(* Logix 5000 project; controller Universal_Device_Info_AOI_V0_1 vendor 1 type 14 code 176 rev 32.11; software revision 32.00; part 3 of 10 *)

           TBEN_L4_8IOL:I.Data[62].11   // IO-Link Port 4 - Input data word 11 (INT bit11)
           TBEN_L4_8IOL:I.Data[62].12   // IO-Link Port 4 - Input data word 11 (INT bit12)
           TBEN_L4_8IOL:I.Data[62].13   // IO-Link Port 4 - Input data word 11 (INT bit13)
           TBEN_L4_8IOL:I.Data[62].14   // IO-Link Port 4 - Input data word 11 (INT bit14)
           TBEN_L4_8IOL:I.Data[62].15   // IO-Link Port 4 - Input data word 11 (INT bit15)
           TBEN_L4_8IOL:I.Data[62].2   // IO-Link Port 4 - Input data word 11 (INT bit2)
           TBEN_L4_8IOL:I.Data[62].3   // IO-Link Port 4 - Input data word 11 (INT bit3)
           TBEN_L4_8IOL:I.Data[62].4   // IO-Link Port 4 - Input data word 11 (INT bit4)
           TBEN_L4_8IOL:I.Data[62].5   // IO-Link Port 4 - Input data word 11 (INT bit5)
           TBEN_L4_8IOL:I.Data[62].6   // IO-Link Port 4 - Input data word 11 (INT bit6)
           TBEN_L4_8IOL:I.Data[62].7   // IO-Link Port 4 - Input data word 11 (INT bit7)
           TBEN_L4_8IOL:I.Data[62].8   // IO-Link Port 4 - Input data word 11 (INT bit8)
           TBEN_L4_8IOL:I.Data[62].9   // IO-Link Port 4 - Input data word 11 (INT bit9)
           TBEN_L4_8IOL:I.Data[63]   // IO-Link Port 4 - Input data word 12
           TBEN_L4_8IOL:I.Data[63].0   // IO-Link Port 4 - Input data word 12 (INT bit0)
           TBEN_L4_8IOL:I.Data[63].1   // IO-Link Port 4 - Input data word 12 (INT bit1)
           TBEN_L4_8IOL:I.Data[63].10   // IO-Link Port 4 - Input data word 12 (INT bit10)
           TBEN_L4_8IOL:I.Data[63].11   // IO-Link Port 4 - Input data word 12 (INT bit11)
           TBEN_L4_8IOL:I.Data[63].12   // IO-Link Port 4 - Input data word 12 (INT bit12)
           TBEN_L4_8IOL:I.Data[63].13   // IO-Link Port 4 - Input data word 12 (INT bit13)
           TBEN_L4_8IOL:I.Data[63].14   // IO-Link Port 4 - Input data word 12 (INT bit14)
           TBEN_L4_8IOL:I.Data[63].15   // IO-Link Port 4 - Input data word 12 (INT bit15)
           TBEN_L4_8IOL:I.Data[63].2   // IO-Link Port 4 - Input data word 12 (INT bit2)
           TBEN_L4_8IOL:I.Data[63].3   // IO-Link Port 4 - Input data word 12 (INT bit3)
           TBEN_L4_8IOL:I.Data[63].4   // IO-Link Port 4 - Input data word 12 (INT bit4)
           TBEN_L4_8IOL:I.Data[63].5   // IO-Link Port 4 - Input data word 12 (INT bit5)
           TBEN_L4_8IOL:I.Data[63].6   // IO-Link Port 4 - Input data word 12 (INT bit6)
           TBEN_L4_8IOL:I.Data[63].7   // IO-Link Port 4 - Input data word 12 (INT bit7)
           TBEN_L4_8IOL:I.Data[63].8   // IO-Link Port 4 - Input data word 12 (INT bit8)
           TBEN_L4_8IOL:I.Data[63].9   // IO-Link Port 4 - Input data word 12 (INT bit9)
           TBEN_L4_8IOL:I.Data[64]   // IO-Link Port 4 - Input data word 13
           TBEN_L4_8IOL:I.Data[64].0   // IO-Link Port 4 - Input data word 13 (INT bit0)
           TBEN_L4_8IOL:I.Data[64].1   // IO-Link Port 4 - Input data word 13 (INT bit1)
           TBEN_L4_8IOL:I.Data[64].10   // IO-Link Port 4 - Input data word 13 (INT bit10)
           TBEN_L4_8IOL:I.Data[64].11   // IO-Link Port 4 - Input data word 13 (INT bit11)
           TBEN_L4_8IOL:I.Data[64].12   // IO-Link Port 4 - Input data word 13 (INT bit12)
           TBEN_L4_8IOL:I.Data[64].13   // IO-Link Port 4 - Input data word 13 (INT bit13)
           TBEN_L4_8IOL:I.Data[64].14   // IO-Link Port 4 - Input data word 13 (INT bit14)
           TBEN_L4_8IOL:I.Data[64].15   // IO-Link Port 4 - Input data word 13 (INT bit15)
           TBEN_L4_8IOL:I.Data[64].2   // IO-Link Port 4 - Input data word 13 (INT bit2)
           TBEN_L4_8IOL:I.Data[64].3   // IO-Link Port 4 - Input data word 13 (INT bit3)
           TBEN_L4_8IOL:I.Data[64].4   // IO-Link Port 4 - Input data word 13 (INT bit4)
           TBEN_L4_8IOL:I.Data[64].5   // IO-Link Port 4 - Input data word 13 (INT bit5)
           TBEN_L4_8IOL:I.Data[64].6   // IO-Link Port 4 - Input data word 13 (INT bit6)
           TBEN_L4_8IOL:I.Data[64].7   // IO-Link Port 4 - Input data word 13 (INT bit7)
           TBEN_L4_8IOL:I.Data[64].8   // IO-Link Port 4 - Input data word 13 (INT bit8)
           TBEN_L4_8IOL:I.Data[64].9   // IO-Link Port 4 - Input data word 13 (INT bit9)
           TBEN_L4_8IOL:I.Data[65]   // IO-Link Port 4 - Input data word 14
           TBEN_L4_8IOL:I.Data[65].0   // IO-Link Port 4 - Input data word 14 (INT bit0)
           TBEN_L4_8IOL:I.Data[65].1   // IO-Link Port 4 - Input data word 14 (INT bit1)
           TBEN_L4_8IOL:I.Data[65].10   // IO-Link Port 4 - Input data word 14 (INT bit10)
           TBEN_L4_8IOL:I.Data[65].11   // IO-Link Port 4 - Input data word 14 (INT bit11)
           TBEN_L4_8IOL:I.Data[65].12   // IO-Link Port 4 - Input data word 14 (INT bit12)
           TBEN_L4_8IOL:I.Data[65].13   // IO-Link Port 4 - Input data word 14 (INT bit13)
           TBEN_L4_8IOL:I.Data[65].14   // IO-Link Port 4 - Input data word 14 (INT bit14)
           TBEN_L4_8IOL:I.Data[65].15   // IO-Link Port 4 - Input data word 14 (INT bit15)
           TBEN_L4_8IOL:I.Data[65].2   // IO-Link Port 4 - Input data word 14 (INT bit2)
           TBEN_L4_8IOL:I.Data[65].3   // IO-Link Port 4 - Input data word 14 (INT bit3)
           TBEN_L4_8IOL:I.Data[65].4   // IO-Link Port 4 - Input data word 14 (INT bit4)
           TBEN_L4_8IOL:I.Data[65].5   // IO-Link Port 4 - Input data word 14 (INT bit5)
           TBEN_L4_8IOL:I.Data[65].6   // IO-Link Port 4 - Input data word 14 (INT bit6)
           TBEN_L4_8IOL:I.Data[65].7   // IO-Link Port 4 - Input data word 14 (INT bit7)
           TBEN_L4_8IOL:I.Data[65].8   // IO-Link Port 4 - Input data word 14 (INT bit8)
           TBEN_L4_8IOL:I.Data[65].9   // IO-Link Port 4 - Input data word 14 (INT bit9)
           TBEN_L4_8IOL:I.Data[66]   // IO-Link Port 4 - Input data word 15
           TBEN_L4_8IOL:I.Data[66].0   // IO-Link Port 4 - Input data word 15 (INT bit0)
           TBEN_L4_8IOL:I.Data[66].1   // IO-Link Port 4 - Input data word 15 (INT bit1)
           TBEN_L4_8IOL:I.Data[66].10   // IO-Link Port 4 - Input data word 15 (INT bit10)
           TBEN_L4_8IOL:I.Data[66].11   // IO-Link Port 4 - Input data word 15 (INT bit11)
           TBEN_L4_8IOL:I.Data[66].12   // IO-Link Port 4 - Input data word 15 (INT bit12)
           TBEN_L4_8IOL:I.Data[66].13   // IO-Link Port 4 - Input data word 15 (INT bit13)
           TBEN_L4_8IOL:I.Data[66].14   // IO-Link Port 4 - Input data word 15 (INT bit14)
           TBEN_L4_8IOL:I.Data[66].15   // IO-Link Port 4 - Input data word 15 (INT bit15)
           TBEN_L4_8IOL:I.Data[66].2   // IO-Link Port 4 - Input data word 15 (INT bit2)
           TBEN_L4_8IOL:I.Data[66].3   // IO-Link Port 4 - Input data word 15 (INT bit3)
           TBEN_L4_8IOL:I.Data[66].4   // IO-Link Port 4 - Input data word 15 (INT bit4)
           TBEN_L4_8IOL:I.Data[66].5   // IO-Link Port 4 - Input data word 15 (INT bit5)
           TBEN_L4_8IOL:I.Data[66].6   // IO-Link Port 4 - Input data word 15 (INT bit6)
           TBEN_L4_8IOL:I.Data[66].7   // IO-Link Port 4 - Input data word 15 (INT bit7)
           TBEN_L4_8IOL:I.Data[66].8   // IO-Link Port 4 - Input data word 15 (INT bit8)
           TBEN_L4_8IOL:I.Data[66].9   // IO-Link Port 4 - Input data word 15 (INT bit9)
           TBEN_L4_8IOL:I.Data[67]   // IO-Link Port 5 - Input data word 0
           TBEN_L4_8IOL:I.Data[67].0   // IO-Link Port 5 - Input data word 0 (INT bit0)
           TBEN_L4_8IOL:I.Data[67].1   // IO-Link Port 5 - Input data word 0 (INT bit1)
           TBEN_L4_8IOL:I.Data[67].10   // IO-Link Port 5 - Input data word 0 (INT bit10)
           TBEN_L4_8IOL:I.Data[67].11   // IO-Link Port 5 - Input data word 0 (INT bit11)
           TBEN_L4_8IOL:I.Data[67].12   // IO-Link Port 5 - Input data word 0 (INT bit12)
           TBEN_L4_8IOL:I.Data[67].13   // IO-Link Port 5 - Input data word 0 (INT bit13)
           TBEN_L4_8IOL:I.Data[67].14   // IO-Link Port 5 - Input data word 0 (INT bit14)
           TBEN_L4_8IOL:I.Data[67].15   // IO-Link Port 5 - Input data word 0 (INT bit15)
           TBEN_L4_8IOL:I.Data[67].2   // IO-Link Port 5 - Input data word 0 (INT bit2)
           TBEN_L4_8IOL:I.Data[67].3   // IO-Link Port 5 - Input data word 0 (INT bit3)
           TBEN_L4_8IOL:I.Data[67].4   // IO-Link Port 5 - Input data word 0 (INT bit4)
           TBEN_L4_8IOL:I.Data[67].5   // IO-Link Port 5 - Input data word 0 (INT bit5)
           TBEN_L4_8IOL:I.Data[67].6   // IO-Link Port 5 - Input data word 0 (INT bit6)
           TBEN_L4_8IOL:I.Data[67].7   // IO-Link Port 5 - Input data word 0 (INT bit7)
           TBEN_L4_8IOL:I.Data[67].8   // IO-Link Port 5 - Input data word 0 (INT bit8)
           TBEN_L4_8IOL:I.Data[67].9   // IO-Link Port 5 - Input data word 0 (INT bit9)
           TBEN_L4_8IOL:I.Data[68]   // IO-Link Port 5 - Input data word 1
           TBEN_L4_8IOL:I.Data[68].0   // IO-Link Port 5 - Input data word 1 (INT bit0)
           TBEN_L4_8IOL:I.Data[68].1   // IO-Link Port 5 - Input data word 1 (INT bit1)
           TBEN_L4_8IOL:I.Data[68].10   // IO-Link Port 5 - Input data word 1 (INT bit10)
           TBEN_L4_8IOL:I.Data[68].11   // IO-Link Port 5 - Input data word 1 (INT bit11)
           TBEN_L4_8IOL:I.Data[68].12   // IO-Link Port 5 - Input data word 1 (INT bit12)
           TBEN_L4_8IOL:I.Data[68].13   // IO-Link Port 5 - Input data word 1 (INT bit13)
           TBEN_L4_8IOL:I.Data[68].14   // IO-Link Port 5 - Input data word 1 (INT bit14)
           TBEN_L4_8IOL:I.Data[68].15   // IO-Link Port 5 - Input data word 1 (INT bit15)
           TBEN_L4_8IOL:I.Data[68].2   // IO-Link Port 5 - Input data word 1 (INT bit2)
           TBEN_L4_8IOL:I.Data[68].3   // IO-Link Port 5 - Input data word 1 (INT bit3)
           TBEN_L4_8IOL:I.Data[68].4   // IO-Link Port 5 - Input data word 1 (INT bit4)
           TBEN_L4_8IOL:I.Data[68].5   // IO-Link Port 5 - Input data word 1 (INT bit5)
           TBEN_L4_8IOL:I.Data[68].6   // IO-Link Port 5 - Input data word 1 (INT bit6)
           TBEN_L4_8IOL:I.Data[68].7   // IO-Link Port 5 - Input data word 1 (INT bit7)
           TBEN_L4_8IOL:I.Data[68].8   // IO-Link Port 5 - Input data word 1 (INT bit8)
           TBEN_L4_8IOL:I.Data[68].9   // IO-Link Port 5 - Input data word 1 (INT bit9)
           TBEN_L4_8IOL:I.Data[69]   // IO-Link Port 5 - Input data word 2
           TBEN_L4_8IOL:I.Data[69].0   // IO-Link Port 5 - Input data word 2 (INT bit0)
           TBEN_L4_8IOL:I.Data[69].1   // IO-Link Port 5 - Input data word 2 (INT bit1)
           TBEN_L4_8IOL:I.Data[69].10   // IO-Link Port 5 - Input data word 2 (INT bit10)
           TBEN_L4_8IOL:I.Data[69].11   // IO-Link Port 5 - Input data word 2 (INT bit11)
           TBEN_L4_8IOL:I.Data[69].12   // IO-Link Port 5 - Input data word 2 (INT bit12)
           TBEN_L4_8IOL:I.Data[69].13   // IO-Link Port 5 - Input data word 2 (INT bit13)
           TBEN_L4_8IOL:I.Data[69].14   // IO-Link Port 5 - Input data word 2 (INT bit14)
           TBEN_L4_8IOL:I.Data[69].15   // IO-Link Port 5 - Input data word 2 (INT bit15)
           TBEN_L4_8IOL:I.Data[69].2   // IO-Link Port 5 - Input data word 2 (INT bit2)
           TBEN_L4_8IOL:I.Data[69].3   // IO-Link Port 5 - Input data word 2 (INT bit3)
           TBEN_L4_8IOL:I.Data[69].4   // IO-Link Port 5 - Input data word 2 (INT bit4)
           TBEN_L4_8IOL:I.Data[69].5   // IO-Link Port 5 - Input data word 2 (INT bit5)
           TBEN_L4_8IOL:I.Data[69].6   // IO-Link Port 5 - Input data word 2 (INT bit6)
           TBEN_L4_8IOL:I.Data[69].7   // IO-Link Port 5 - Input data word 2 (INT bit7)
           TBEN_L4_8IOL:I.Data[69].8   // IO-Link Port 5 - Input data word 2 (INT bit8)
           TBEN_L4_8IOL:I.Data[69].9   // IO-Link Port 5 - Input data word 2 (INT bit9)
           TBEN_L4_8IOL:I.Data[6]   // IO-Link Port 1 - Input data word 3
           TBEN_L4_8IOL:I.Data[6].0   // IO-Link Port 1 - Input data word 3 (INT bit0)
           TBEN_L4_8IOL:I.Data[6].1   // IO-Link Port 1 - Input data word 3 (INT bit1)
           TBEN_L4_8IOL:I.Data[6].10   // IO-Link Port 1 - Input data word 3 (INT bit10)
           TBEN_L4_8IOL:I.Data[6].11   // IO-Link Port 1 - Input data word 3 (INT bit11)
           TBEN_L4_8IOL:I.Data[6].12   // IO-Link Port 1 - Input data word 3 (INT bit12)
           TBEN_L4_8IOL:I.Data[6].13   // IO-Link Port 1 - Input data word 3 (INT bit13)
           TBEN_L4_8IOL:I.Data[6].14   // IO-Link Port 1 - Input data word 3 (INT bit14)
           TBEN_L4_8IOL:I.Data[6].15   // IO-Link Port 1 - Input data word 3 (INT bit15)
           TBEN_L4_8IOL:I.Data[6].2   // IO-Link Port 1 - Input data word 3 (INT bit2)
           TBEN_L4_8IOL:I.Data[6].3   // IO-Link Port 1 - Input data word 3 (INT bit3)
           TBEN_L4_8IOL:I.Data[6].4   // IO-Link Port 1 - Input data word 3 (INT bit4)
           TBEN_L4_8IOL:I.Data[6].5   // IO-Link Port 1 - Input data word 3 (INT bit5)
           TBEN_L4_8IOL:I.Data[6].6   // IO-Link Port 1 - Input data word 3 (INT bit6)
           TBEN_L4_8IOL:I.Data[6].7   // IO-Link Port 1 - Input data word 3 (INT bit7)
           TBEN_L4_8IOL:I.Data[6].8   // IO-Link Port 1 - Input data word 3 (INT bit8)
           TBEN_L4_8IOL:I.Data[6].9   // IO-Link Port 1 - Input data word 3 (INT bit9)
           TBEN_L4_8IOL:I.Data[70]   // IO-Link Port 5 - Input data word 3
           TBEN_L4_8IOL:I.Data[70].0   // IO-Link Port 5 - Input data word 3 (INT bit0)
           TBEN_L4_8IOL:I.Data[70].1   // IO-Link Port 5 - Input data word 3 (INT bit1)
           TBEN_L4_8IOL:I.Data[70].10   // IO-Link Port 5 - Input data word 3 (INT bit10)
           TBEN_L4_8IOL:I.Data[70].11   // IO-Link Port 5 - Input data word 3 (INT bit11)
           TBEN_L4_8IOL:I.Data[70].12   // IO-Link Port 5 - Input data word 3 (INT bit12)
           TBEN_L4_8IOL:I.Data[70].13   // IO-Link Port 5 - Input data word 3 (INT bit13)
           TBEN_L4_8IOL:I.Data[70].14   // IO-Link Port 5 - Input data word 3 (INT bit14)
           TBEN_L4_8IOL:I.Data[70].15   // IO-Link Port 5 - Input data word 3 (INT bit15)
           TBEN_L4_8IOL:I.Data[70].2   // IO-Link Port 5 - Input data word 3 (INT bit2)
           TBEN_L4_8IOL:I.Data[70].3   // IO-Link Port 5 - Input data word 3 (INT bit3)
           TBEN_L4_8IOL:I.Data[70].4   // IO-Link Port 5 - Input data word 3 (INT bit4)
           TBEN_L4_8IOL:I.Data[70].5   // IO-Link Port 5 - Input data word 3 (INT bit5)
           TBEN_L4_8IOL:I.Data[70].6   // IO-Link Port 5 - Input data word 3 (INT bit6)
           TBEN_L4_8IOL:I.Data[70].7   // IO-Link Port 5 - Input data word 3 (INT bit7)
           TBEN_L4_8IOL:I.Data[70].8   // IO-Link Port 5 - Input data word 3 (INT bit8)
           TBEN_L4_8IOL:I.Data[70].9   // IO-Link Port 5 - Input data word 3 (INT bit9)
           TBEN_L4_8IOL:I.Data[71]   // IO-Link Port 5 - Input data word 4
           TBEN_L4_8IOL:I.Data[71].0   // IO-Link Port 5 - Input data word 4 (INT bit0)
           TBEN_L4_8IOL:I.Data[71].1   // IO-Link Port 5 - Input data word 4 (INT bit1)
           TBEN_L4_8IOL:I.Data[71].10   // IO-Link Port 5 - Input data word 4 (INT bit10)
           TBEN_L4_8IOL:I.Data[71].11   // IO-Link Port 5 - Input data word 4 (INT bit11)
           TBEN_L4_8IOL:I.Data[71].12   // IO-Link Port 5 - Input data word 4 (INT bit12)
           TBEN_L4_8IOL:I.Data[71].13   // IO-Link Port 5 - Input data word 4 (INT bit13)
           TBEN_L4_8IOL:I.Data[71].14   // IO-Link Port 5 - Input data word 4 (INT bit14)
           TBEN_L4_8IOL:I.Data[71].15   // IO-Link Port 5 - Input data word 4 (INT bit15)
           TBEN_L4_8IOL:I.Data[71].2   // IO-Link Port 5 - Input data word 4 (INT bit2)
           TBEN_L4_8IOL:I.Data[71].3   // IO-Link Port 5 - Input data word 4 (INT bit3)
           TBEN_L4_8IOL:I.Data[71].4   // IO-Link Port 5 - Input data word 4 (INT bit4)
           TBEN_L4_8IOL:I.Data[71].5   // IO-Link Port 5 - Input data word 4 (INT bit5)
           TBEN_L4_8IOL:I.Data[71].6   // IO-Link Port 5 - Input data word 4 (INT bit6)
           TBEN_L4_8IOL:I.Data[71].7   // IO-Link Port 5 - Input data word 4 (INT bit7)
           TBEN_L4_8IOL:I.Data[71].8   // IO-Link Port 5 - Input data word 4 (INT bit8)
           TBEN_L4_8IOL:I.Data[71].9   // IO-Link Port 5 - Input data word 4 (INT bit9)
           TBEN_L4_8IOL:I.Data[72]   // IO-Link Port 5 - Input data word 5
           TBEN_L4_8IOL:I.Data[72].0   // IO-Link Port 5 - Input data word 5 (INT bit0)
           TBEN_L4_8IOL:I.Data[72].1   // IO-Link Port 5 - Input data word 5 (INT bit1)
           TBEN_L4_8IOL:I.Data[72].10   // IO-Link Port 5 - Input data word 5 (INT bit10)
           TBEN_L4_8IOL:I.Data[72].11   // IO-Link Port 5 - Input data word 5 (INT bit11)
           TBEN_L4_8IOL:I.Data[72].12   // IO-Link Port 5 - Input data word 5 (INT bit12)
           TBEN_L4_8IOL:I.Data[72].13   // IO-Link Port 5 - Input data word 5 (INT bit13)
           TBEN_L4_8IOL:I.Data[72].14   // IO-Link Port 5 - Input data word 5 (INT bit14)
           TBEN_L4_8IOL:I.Data[72].15   // IO-Link Port 5 - Input data word 5 (INT bit15)
           TBEN_L4_8IOL:I.Data[72].2   // IO-Link Port 5 - Input data word 5 (INT bit2)
           TBEN_L4_8IOL:I.Data[72].3   // IO-Link Port 5 - Input data word 5 (INT bit3)
           TBEN_L4_8IOL:I.Data[72].4   // IO-Link Port 5 - Input data word 5 (INT bit4)
           TBEN_L4_8IOL:I.Data[72].5   // IO-Link Port 5 - Input data word 5 (INT bit5)
           TBEN_L4_8IOL:I.Data[72].6   // IO-Link Port 5 - Input data word 5 (INT bit6)
           TBEN_L4_8IOL:I.Data[72].7   // IO-Link Port 5 - Input data word 5 (INT bit7)
           TBEN_L4_8IOL:I.Data[72].8   // IO-Link Port 5 - Input data word 5 (INT bit8)
           TBEN_L4_8IOL:I.Data[72].9   // IO-Link Port 5 - Input data word 5 (INT bit9)
           TBEN_L4_8IOL:I.Data[73]   // IO-Link Port 5 - Input data word 6
           TBEN_L4_8IOL:I.Data[73].0   // IO-Link Port 5 - Input data word 6 (INT bit0)
           TBEN_L4_8IOL:I.Data[73].1   // IO-Link Port 5 - Input data word 6 (INT bit1)
           TBEN_L4_8IOL:I.Data[73].10   // IO-Link Port 5 - Input data word 6 (INT bit10)
           TBEN_L4_8IOL:I.Data[73].11   // IO-Link Port 5 - Input data word 6 (INT bit11)
           TBEN_L4_8IOL:I.Data[73].12   // IO-Link Port 5 - Input data word 6 (INT bit12)
           TBEN_L4_8IOL:I.Data[73].13   // IO-Link Port 5 - Input data word 6 (INT bit13)
           TBEN_L4_8IOL:I.Data[73].14   // IO-Link Port 5 - Input data word 6 (INT bit14)
           TBEN_L4_8IOL:I.Data[73].15   // IO-Link Port 5 - Input data word 6 (INT bit15)
           TBEN_L4_8IOL:I.Data[73].2   // IO-Link Port 5 - Input data word 6 (INT bit2)
           TBEN_L4_8IOL:I.Data[73].3   // IO-Link Port 5 - Input data word 6 (INT bit3)
           TBEN_L4_8IOL:I.Data[73].4   // IO-Link Port 5 - Input data word 6 (INT bit4)
           TBEN_L4_8IOL:I.Data[73].5   // IO-Link Port 5 - Input data word 6 (INT bit5)
           TBEN_L4_8IOL:I.Data[73].6   // IO-Link Port 5 - Input data word 6 (INT bit6)
           TBEN_L4_8IOL:I.Data[73].7   // IO-Link Port 5 - Input data word 6 (INT bit7)
           TBEN_L4_8IOL:I.Data[73].8   // IO-Link Port 5 - Input data word 6 (INT bit8)
           TBEN_L4_8IOL:I.Data[73].9   // IO-Link Port 5 - Input data word 6 (INT bit9)
           TBEN_L4_8IOL:I.Data[74]   // IO-Link Port 5 - Input data word 7
           TBEN_L4_8IOL:I.Data[74].0   // IO-Link Port 5 - Input data word 7 (INT bit0)
           TBEN_L4_8IOL:I.Data[74].1   // IO-Link Port 5 - Input data word 7 (INT bit1)
           TBEN_L4_8IOL:I.Data[74].10   // IO-Link Port 5 - Input data word 7 (INT bit10)
           TBEN_L4_8IOL:I.Data[74].11   // IO-Link Port 5 - Input data word 7 (INT bit11)
           TBEN_L4_8IOL:I.Data[74].12   // IO-Link Port 5 - Input data word 7 (INT bit12)
           TBEN_L4_8IOL:I.Data[74].13   // IO-Link Port 5 - Input data word 7 (INT bit13)
           TBEN_L4_8IOL:I.Data[74].14   // IO-Link Port 5 - Input data word 7 (INT bit14)
           TBEN_L4_8IOL:I.Data[74].15   // IO-Link Port 5 - Input data word 7 (INT bit15)
           TBEN_L4_8IOL:I.Data[74].2   // IO-Link Port 5 - Input data word 7 (INT bit2)
           TBEN_L4_8IOL:I.Data[74].3   // IO-Link Port 5 - Input data word 7 (INT bit3)
           TBEN_L4_8IOL:I.Data[74].4   // IO-Link Port 5 - Input data word 7 (INT bit4)
           TBEN_L4_8IOL:I.Data[74].5   // IO-Link Port 5 - Input data word 7 (INT bit5)
           TBEN_L4_8IOL:I.Data[74].6   // IO-Link Port 5 - Input data word 7 (INT bit6)
           TBEN_L4_8IOL:I.Data[74].7   // IO-Link Port 5 - Input data word 7 (INT bit7)
           TBEN_L4_8IOL:I.Data[74].8   // IO-Link Port 5 - Input data word 7 (INT bit8)
           TBEN_L4_8IOL:I.Data[74].9   // IO-Link Port 5 - Input data word 7 (INT bit9)
           TBEN_L4_8IOL:I.Data[75]   // IO-Link Port 5 - Input data word 8
           TBEN_L4_8IOL:I.Data[75].0   // IO-Link Port 5 - Input data word 8 (INT bit0)
           TBEN_L4_8IOL:I.Data[75].1   // IO-Link Port 5 - Input data word 8 (INT bit1)
           TBEN_L4_8IOL:I.Data[75].10   // IO-Link Port 5 - Input data word 8 (INT bit10)
           TBEN_L4_8IOL:I.Data[75].11   // IO-Link Port 5 - Input data word 8 (INT bit11)
           TBEN_L4_8IOL:I.Data[75].12   // IO-Link Port 5 - Input data word 8 (INT bit12)
           TBEN_L4_8IOL:I.Data[75].13   // IO-Link Port 5 - Input data word 8 (INT bit13)
           TBEN_L4_8IOL:I.Data[75].14   // IO-Link Port 5 - Input data word 8 (INT bit14)
           TBEN_L4_8IOL:I.Data[75].15   // IO-Link Port 5 - Input data word 8 (INT bit15)
           TBEN_L4_8IOL:I.Data[75].2   // IO-Link Port 5 - Input data word 8 (INT bit2)
           TBEN_L4_8IOL:I.Data[75].3   // IO-Link Port 5 - Input data word 8 (INT bit3)
           TBEN_L4_8IOL:I.Data[75].4   // IO-Link Port 5 - Input data word 8 (INT bit4)
           TBEN_L4_8IOL:I.Data[75].5   // IO-Link Port 5 - Input data word 8 (INT bit5)
           TBEN_L4_8IOL:I.Data[75].6   // IO-Link Port 5 - Input data word 8 (INT bit6)
           TBEN_L4_8IOL:I.Data[75].7   // IO-Link Port 5 - Input data word 8 (INT bit7)
           TBEN_L4_8IOL:I.Data[75].8   // IO-Link Port 5 - Input data word 8 (INT bit8)
           TBEN_L4_8IOL:I.Data[75].9   // IO-Link Port 5 - Input data word 8 (INT bit9)
           TBEN_L4_8IOL:I.Data[76]   // IO-Link Port 5 - Input data word 9
           TBEN_L4_8IOL:I.Data[76].0   // IO-Link Port 5 - Input data word 9 (INT bit0)
           TBEN_L4_8IOL:I.Data[76].1   // IO-Link Port 5 - Input data word 9 (INT bit1)
           TBEN_L4_8IOL:I.Data[76].10   // IO-Link Port 5 - Input data word 9 (INT bit10)
           TBEN_L4_8IOL:I.Data[76].11   // IO-Link Port 5 - Input data word 9 (INT bit11)
           TBEN_L4_8IOL:I.Data[76].12   // IO-Link Port 5 - Input data word 9 (INT bit12)
           TBEN_L4_8IOL:I.Data[76].13   // IO-Link Port 5 - Input data word 9 (INT bit13)
           TBEN_L4_8IOL:I.Data[76].14   // IO-Link Port 5 - Input data word 9 (INT bit14)
           TBEN_L4_8IOL:I.Data[76].15   // IO-Link Port 5 - Input data word 9 (INT bit15)
           TBEN_L4_8IOL:I.Data[76].2   // IO-Link Port 5 - Input data word 9 (INT bit2)
           TBEN_L4_8IOL:I.Data[76].3   // IO-Link Port 5 - Input data word 9 (INT bit3)
           TBEN_L4_8IOL:I.Data[76].4   // IO-Link Port 5 - Input data word 9 (INT bit4)
           TBEN_L4_8IOL:I.Data[76].5   // IO-Link Port 5 - Input data word 9 (INT bit5)
           TBEN_L4_8IOL:I.Data[76].6   // IO-Link Port 5 - Input data word 9 (INT bit6)
           TBEN_L4_8IOL:I.Data[76].7   // IO-Link Port 5 - Input data word 9 (INT bit7)
           TBEN_L4_8IOL:I.Data[76].8   // IO-Link Port 5 - Input data word 9 (INT bit8)
           TBEN_L4_8IOL:I.Data[76].9   // IO-Link Port 5 - Input data word 9 (INT bit9)
           TBEN_L4_8IOL:I.Data[77]   // IO-Link Port 5 - Input data word 10
           TBEN_L4_8IOL:I.Data[77].0   // IO-Link Port 5 - Input data word 10 (INT bit0)
           TBEN_L4_8IOL:I.Data[77].1   // IO-Link Port 5 - Input data word 10 (INT bit1)
           TBEN_L4_8IOL:I.Data[77].10   // IO-Link Port 5 - Input data word 10 (INT bit10)
           TBEN_L4_8IOL:I.Data[77].11   // IO-Link Port 5 - Input data word 10 (INT bit11)
           TBEN_L4_8IOL:I.Data[77].12   // IO-Link Port 5 - Input data word 10 (INT bit12)
           TBEN_L4_8IOL:I.Data[77].13   // IO-Link Port 5 - Input data word 10 (INT bit13)
           TBEN_L4_8IOL:I.Data[77].14   // IO-Link Port 5 - Input data word 10 (INT bit14)
           TBEN_L4_8IOL:I.Data[77].15   // IO-Link Port 5 - Input data word 10 (INT bit15)
           TBEN_L4_8IOL:I.Data[77].2   // IO-Link Port 5 - Input data word 10 (INT bit2)
           TBEN_L4_8IOL:I.Data[77].3   // IO-Link Port 5 - Input data word 10 (INT bit3)
           TBEN_L4_8IOL:I.Data[77].4   // IO-Link Port 5 - Input data word 10 (INT bit4)
           TBEN_L4_8IOL:I.Data[77].5   // IO-Link Port 5 - Input data word 10 (INT bit5)
           TBEN_L4_8IOL:I.Data[77].6   // IO-Link Port 5 - Input data word 10 (INT bit6)
           TBEN_L4_8IOL:I.Data[77].7   // IO-Link Port 5 - Input data word 10 (INT bit7)
           TBEN_L4_8IOL:I.Data[77].8   // IO-Link Port 5 - Input data word 10 (INT bit8)
           TBEN_L4_8IOL:I.Data[77].9   // IO-Link Port 5 - Input data word 10 (INT bit9)
           TBEN_L4_8IOL:I.Data[78]   // IO-Link Port 5 - Input data word 11
           TBEN_L4_8IOL:I.Data[78].0   // IO-Link Port 5 - Input data word 11 (INT bit0)
           TBEN_L4_8IOL:I.Data[78].1   // IO-Link Port 5 - Input data word 11 (INT bit1)
           TBEN_L4_8IOL:I.Data[78].10   // IO-Link Port 5 - Input data word 11 (INT bit10)
           TBEN_L4_8IOL:I.Data[78].11   // IO-Link Port 5 - Input data word 11 (INT bit11)
           TBEN_L4_8IOL:I.Data[78].12   // IO-Link Port 5 - Input data word 11 (INT bit12)
           TBEN_L4_8IOL:I.Data[78].13   // IO-Link Port 5 - Input data word 11 (INT bit13)
           TBEN_L4_8IOL:I.Data[78].14   // IO-Link Port 5 - Input data word 11 (INT bit14)
           TBEN_L4_8IOL:I.Data[78].15   // IO-Link Port 5 - Input data word 11 (INT bit15)
           TBEN_L4_8IOL:I.Data[78].2   // IO-Link Port 5 - Input data word 11 (INT bit2)
           TBEN_L4_8IOL:I.Data[78].3   // IO-Link Port 5 - Input data word 11 (INT bit3)
           TBEN_L4_8IOL:I.Data[78].4   // IO-Link Port 5 - Input data word 11 (INT bit4)
           TBEN_L4_8IOL:I.Data[78].5   // IO-Link Port 5 - Input data word 11 (INT bit5)
           TBEN_L4_8IOL:I.Data[78].6   // IO-Link Port 5 - Input data word 11 (INT bit6)
           TBEN_L4_8IOL:I.Data[78].7   // IO-Link Port 5 - Input data word 11 (INT bit7)
           TBEN_L4_8IOL:I.Data[78].8   // IO-Link Port 5 - Input data word 11 (INT bit8)
           TBEN_L4_8IOL:I.Data[78].9   // IO-Link Port 5 - Input data word 11 (INT bit9)
           TBEN_L4_8IOL:I.Data[79]   // IO-Link Port 5 - Input data word 12
           TBEN_L4_8IOL:I.Data[79].0   // IO-Link Port 5 - Input data word 12 (INT bit0)
           TBEN_L4_8IOL:I.Data[79].1   // IO-Link Port 5 - Input data word 12 (INT bit1)
           TBEN_L4_8IOL:I.Data[79].10   // IO-Link Port 5 - Input data word 12 (INT bit10)
           TBEN_L4_8IOL:I.Data[79].11   // IO-Link Port 5 - Input data word 12 (INT bit11)
           TBEN_L4_8IOL:I.Data[79].12   // IO-Link Port 5 - Input data word 12 (INT bit12)
           TBEN_L4_8IOL:I.Data[79].13   // IO-Link Port 5 - Input data word 12 (INT bit13)
           TBEN_L4_8IOL:I.Data[79].14   // IO-Link Port 5 - Input data word 12 (INT bit14)
           TBEN_L4_8IOL:I.Data[79].15   // IO-Link Port 5 - Input data word 12 (INT bit15)
           TBEN_L4_8IOL:I.Data[79].2   // IO-Link Port 5 - Input data word 12 (INT bit2)
           TBEN_L4_8IOL:I.Data[79].3   // IO-Link Port 5 - Input data word 12 (INT bit3)
           TBEN_L4_8IOL:I.Data[79].4   // IO-Link Port 5 - Input data word 12 (INT bit4)
           TBEN_L4_8IOL:I.Data[79].5   // IO-Link Port 5 - Input data word 12 (INT bit5)
           TBEN_L4_8IOL:I.Data[79].6   // IO-Link Port 5 - Input data word 12 (INT bit6)
           TBEN_L4_8IOL:I.Data[79].7   // IO-Link Port 5 - Input data word 12 (INT bit7)
           TBEN_L4_8IOL:I.Data[79].8   // IO-Link Port 5 - Input data word 12 (INT bit8)
           TBEN_L4_8IOL:I.Data[79].9   // IO-Link Port 5 - Input data word 12 (INT bit9)
           TBEN_L4_8IOL:I.Data[7]   // IO-Link Port 1 - Input data word 4
           TBEN_L4_8IOL:I.Data[7].0   // IO-Link Port 1 - Input data word 4 (INT bit0)
           TBEN_L4_8IOL:I.Data[7].1   // IO-Link Port 1 - Input data word 4 (INT bit1)
           TBEN_L4_8IOL:I.Data[7].10   // IO-Link Port 1 - Input data word 4 (INT bit10)
           TBEN_L4_8IOL:I.Data[7].11   // IO-Link Port 1 - Input data word 4 (INT bit11)
           TBEN_L4_8IOL:I.Data[7].12   // IO-Link Port 1 - Input data word 4 (INT bit12)
           TBEN_L4_8IOL:I.Data[7].13   // IO-Link Port 1 - Input data word 4 (INT bit13)
           TBEN_L4_8IOL:I.Data[7].14   // IO-Link Port 1 - Input data word 4 (INT bit14)
           TBEN_L4_8IOL:I.Data[7].15   // IO-Link Port 1 - Input data word 4 (INT bit15)
           TBEN_L4_8IOL:I.Data[7].2   // IO-Link Port 1 - Input data word 4 (INT bit2)
           TBEN_L4_8IOL:I.Data[7].3   // IO-Link Port 1 - Input data word 4 (INT bit3)
           TBEN_L4_8IOL:I.Data[7].4   // IO-Link Port 1 - Input data word 4 (INT bit4)
           TBEN_L4_8IOL:I.Data[7].5   // IO-Link Port 1 - Input data word 4 (INT bit5)
           TBEN_L4_8IOL:I.Data[7].6   // IO-Link Port 1 - Input data word 4 (INT bit6)
           TBEN_L4_8IOL:I.Data[7].7   // IO-Link Port 1 - Input data word 4 (INT bit7)
           TBEN_L4_8IOL:I.Data[7].8   // IO-Link Port 1 - Input data word 4 (INT bit8)
           TBEN_L4_8IOL:I.Data[7].9   // IO-Link Port 1 - Input data word 4 (INT bit9)
           TBEN_L4_8IOL:I.Data[80]   // IO-Link Port 5 - Input data word 13
           TBEN_L4_8IOL:I.Data[80].0   // IO-Link Port 5 - Input data word 13 (INT bit0)
           TBEN_L4_8IOL:I.Data[80].1   // IO-Link Port 5 - Input data word 13 (INT bit1)
           TBEN_L4_8IOL:I.Data[80].10   // IO-Link Port 5 - Input data word 13 (INT bit10)
           TBEN_L4_8IOL:I.Data[80].11   // IO-Link Port 5 - Input data word 13 (INT bit11)
           TBEN_L4_8IOL:I.Data[80].12   // IO-Link Port 5 - Input data word 13 (INT bit12)
           TBEN_L4_8IOL:I.Data[80].13   // IO-Link Port 5 - Input data word 13 (INT bit13)
           TBEN_L4_8IOL:I.Data[80].14   // IO-Link Port 5 - Input data word 13 (INT bit14)
           TBEN_L4_8IOL:I.Data[80].15   // IO-Link Port 5 - Input data word 13 (INT bit15)
           TBEN_L4_8IOL:I.Data[80].2   // IO-Link Port 5 - Input data word 13 (INT bit2)
           TBEN_L4_8IOL:I.Data[80].3   // IO-Link Port 5 - Input data word 13 (INT bit3)
           TBEN_L4_8IOL:I.Data[80].4   // IO-Link Port 5 - Input data word 13 (INT bit4)
           TBEN_L4_8IOL:I.Data[80].5   // IO-Link Port 5 - Input data word 13 (INT bit5)
           TBEN_L4_8IOL:I.Data[80].6   // IO-Link Port 5 - Input data word 13 (INT bit6)
           TBEN_L4_8IOL:I.Data[80].7   // IO-Link Port 5 - Input data word 13 (INT bit7)
           TBEN_L4_8IOL:I.Data[80].8   // IO-Link Port 5 - Input data word 13 (INT bit8)
           TBEN_L4_8IOL:I.Data[80].9   // IO-Link Port 5 - Input data word 13 (INT bit9)
           TBEN_L4_8IOL:I.Data[81]   // IO-Link Port 5 - Input data word 14
           TBEN_L4_8IOL:I.Data[81].0   // IO-Link Port 5 - Input data word 14 (INT bit0)
           TBEN_L4_8IOL:I.Data[81].1   // IO-Link Port 5 - Input data word 14 (INT bit1)
           TBEN_L4_8IOL:I.Data[81].10   // IO-Link Port 5 - Input data word 14 (INT bit10)
           TBEN_L4_8IOL:I.Data[81].11   // IO-Link Port 5 - Input data word 14 (INT bit11)
           TBEN_L4_8IOL:I.Data[81].12   // IO-Link Port 5 - Input data word 14 (INT bit12)
           TBEN_L4_8IOL:I.Data[81].13   // IO-Link Port 5 - Input data word 14 (INT bit13)
           TBEN_L4_8IOL:I.Data[81].14   // IO-Link Port 5 - Input data word 14 (INT bit14)
           TBEN_L4_8IOL:I.Data[81].15   // IO-Link Port 5 - Input data word 14 (INT bit15)
           TBEN_L4_8IOL:I.Data[81].2   // IO-Link Port 5 - Input data word 14 (INT bit2)
           TBEN_L4_8IOL:I.Data[81].3   // IO-Link Port 5 - Input data word 14 (INT bit3)
           TBEN_L4_8IOL:I.Data[81].4   // IO-Link Port 5 - Input data word 14 (INT bit4)
           TBEN_L4_8IOL:I.Data[81].5   // IO-Link Port 5 - Input data word 14 (INT bit5)
           TBEN_L4_8IOL:I.Data[81].6   // IO-Link Port 5 - Input data word 14 (INT bit6)
           TBEN_L4_8IOL:I.Data[81].7   // IO-Link Port 5 - Input data word 14 (INT bit7)
           TBEN_L4_8IOL:I.Data[81].8   // IO-Link Port 5 - Input data word 14 (INT bit8)
           TBEN_L4_8IOL:I.Data[81].9   // IO-Link Port 5 - Input data word 14 (INT bit9)
           TBEN_L4_8IOL:I.Data[82]   // IO-Link Port 5 - Input data word 15
           TBEN_L4_8IOL:I.Data[82].0   // IO-Link Port 5 - Input data word 15 (INT bit0)
           TBEN_L4_8IOL:I.Data[82].1   // IO-Link Port 5 - Input data word 15 (INT bit1)
           TBEN_L4_8IOL:I.Data[82].10   // IO-Link Port 5 - Input data word 15 (INT bit10)
           TBEN_L4_8IOL:I.Data[82].11   // IO-Link Port 5 - Input data word 15 (INT bit11)
           TBEN_L4_8IOL:I.Data[82].12   // IO-Link Port 5 - Input data word 15 (INT bit12)
           TBEN_L4_8IOL:I.Data[82].13   // IO-Link Port 5 - Input data word 15 (INT bit13)
           TBEN_L4_8IOL:I.Data[82].14   // IO-Link Port 5 - Input data word 15 (INT bit14)
           TBEN_L4_8IOL:I.Data[82].15   // IO-Link Port 5 - Input data word 15 (INT bit15)
           TBEN_L4_8IOL:I.Data[82].2   // IO-Link Port 5 - Input data word 15 (INT bit2)
           TBEN_L4_8IOL:I.Data[82].3   // IO-Link Port 5 - Input data word 15 (INT bit3)
           TBEN_L4_8IOL:I.Data[82].4   // IO-Link Port 5 - Input data word 15 (INT bit4)
           TBEN_L4_8IOL:I.Data[82].5   // IO-Link Port 5 - Input data word 15 (INT bit5)
           TBEN_L4_8IOL:I.Data[82].6   // IO-Link Port 5 - Input data word 15 (INT bit6)
           TBEN_L4_8IOL:I.Data[82].7   // IO-Link Port 5 - Input data word 15 (INT bit7)
           TBEN_L4_8IOL:I.Data[82].8   // IO-Link Port 5 - Input data word 15 (INT bit8)
           TBEN_L4_8IOL:I.Data[82].9   // IO-Link Port 5 - Input data word 15 (INT bit9)
           TBEN_L4_8IOL:I.Data[83]   // IO-Link Port 6 - Input data word 0
           TBEN_L4_8IOL:I.Data[83].0   // IO-Link Port 6 - Input data word 0 (INT bit0)
           TBEN_L4_8IOL:I.Data[83].1   // IO-Link Port 6 - Input data word 0 (INT bit1)
           TBEN_L4_8IOL:I.Data[83].10   // IO-Link Port 6 - Input data word 0 (INT bit10)
           TBEN_L4_8IOL:I.Data[83].11   // IO-Link Port 6 - Input data word 0 (INT bit11)
           TBEN_L4_8IOL:I.Data[83].12   // IO-Link Port 6 - Input data word 0 (INT bit12)
           TBEN_L4_8IOL:I.Data[83].13   // IO-Link Port 6 - Input data word 0 (INT bit13)
           TBEN_L4_8IOL:I.Data[83].14   // IO-Link Port 6 - Input data word 0 (INT bit14)
           TBEN_L4_8IOL:I.Data[83].15   // IO-Link Port 6 - Input data word 0 (INT bit15)
           TBEN_L4_8IOL:I.Data[83].2   // IO-Link Port 6 - Input data word 0 (INT bit2)
           TBEN_L4_8IOL:I.Data[83].3   // IO-Link Port 6 - Input data word 0 (INT bit3)
           TBEN_L4_8IOL:I.Data[83].4   // IO-Link Port 6 - Input data word 0 (INT bit4)
           TBEN_L4_8IOL:I.Data[83].5   // IO-Link Port 6 - Input data word 0 (INT bit5)
           TBEN_L4_8IOL:I.Data[83].6   // IO-Link Port 6 - Input data word 0 (INT bit6)
           TBEN_L4_8IOL:I.Data[83].7   // IO-Link Port 6 - Input data word 0 (INT bit7)
           TBEN_L4_8IOL:I.Data[83].8   // IO-Link Port 6 - Input data word 0 (INT bit8)
           TBEN_L4_8IOL:I.Data[83].9   // IO-Link Port 6 - Input data word 0 (INT bit9)
           TBEN_L4_8IOL:I.Data[84]   // IO-Link Port 6 - Input data word 1
           TBEN_L4_8IOL:I.Data[84].0   // IO-Link Port 6 - Input data word 1 (INT bit0)
           TBEN_L4_8IOL:I.Data[84].1   // IO-Link Port 6 - Input data word 1 (INT bit1)
           TBEN_L4_8IOL:I.Data[84].10   // IO-Link Port 6 - Input data word 1 (INT bit10)
           TBEN_L4_8IOL:I.Data[84].11   // IO-Link Port 6 - Input data word 1 (INT bit11)
           TBEN_L4_8IOL:I.Data[84].12   // IO-Link Port 6 - Input data word 1 (INT bit12)
           TBEN_L4_8IOL:I.Data[84].13   // IO-Link Port 6 - Input data word 1 (INT bit13)
           TBEN_L4_8IOL:I.Data[84].14   // IO-Link Port 6 - Input data word 1 (INT bit14)
           TBEN_L4_8IOL:I.Data[84].15   // IO-Link Port 6 - Input data word 1 (INT bit15)
           TBEN_L4_8IOL:I.Data[84].2   // IO-Link Port 6 - Input data word 1 (INT bit2)
           TBEN_L4_8IOL:I.Data[84].3   // IO-Link Port 6 - Input data word 1 (INT bit3)
           TBEN_L4_8IOL:I.Data[84].4   // IO-Link Port 6 - Input data word 1 (INT bit4)
           TBEN_L4_8IOL:I.Data[84].5   // IO-Link Port 6 - Input data word 1 (INT bit5)
           TBEN_L4_8IOL:I.Data[84].6   // IO-Link Port 6 - Input data word 1 (INT bit6)
           TBEN_L4_8IOL:I.Data[84].7   // IO-Link Port 6 - Input data word 1 (INT bit7)
           TBEN_L4_8IOL:I.Data[84].8   // IO-Link Port 6 - Input data word 1 (INT bit8)
           TBEN_L4_8IOL:I.Data[84].9   // IO-Link Port 6 - Input data word 1 (INT bit9)
           TBEN_L4_8IOL:I.Data[85]   // IO-Link Port 6 - Input data word 2
           TBEN_L4_8IOL:I.Data[85].0   // IO-Link Port 6 - Input data word 2 (INT bit0)
           TBEN_L4_8IOL:I.Data[85].1   // IO-Link Port 6 - Input data word 2 (INT bit1)
           TBEN_L4_8IOL:I.Data[85].10   // IO-Link Port 6 - Input data word 2 (INT bit10)
           TBEN_L4_8IOL:I.Data[85].11   // IO-Link Port 6 - Input data word 2 (INT bit11)
           TBEN_L4_8IOL:I.Data[85].12   // IO-Link Port 6 - Input data word 2 (INT bit12)
           TBEN_L4_8IOL:I.Data[85].13   // IO-Link Port 6 - Input data word 2 (INT bit13)
           TBEN_L4_8IOL:I.Data[85].14   // IO-Link Port 6 - Input data word 2 (INT bit14)
           TBEN_L4_8IOL:I.Data[85].15   // IO-Link Port 6 - Input data word 2 (INT bit15)
           TBEN_L4_8IOL:I.Data[85].2   // IO-Link Port 6 - Input data word 2 (INT bit2)
           TBEN_L4_8IOL:I.Data[85].3   // IO-Link Port 6 - Input data word 2 (INT bit3)
           TBEN_L4_8IOL:I.Data[85].4   // IO-Link Port 6 - Input data word 2 (INT bit4)
           TBEN_L4_8IOL:I.Data[85].5   // IO-Link Port 6 - Input data word 2 (INT bit5)
           TBEN_L4_8IOL:I.Data[85].6   // IO-Link Port 6 - Input data word 2 (INT bit6)
           TBEN_L4_8IOL:I.Data[85].7   // IO-Link Port 6 - Input data word 2 (INT bit7)
           TBEN_L4_8IOL:I.Data[85].8   // IO-Link Port 6 - Input data word 2 (INT bit8)
           TBEN_L4_8IOL:I.Data[85].9   // IO-Link Port 6 - Input data word 2 (INT bit9)
           TBEN_L4_8IOL:I.Data[86]   // IO-Link Port 6 - Input data word 3
           TBEN_L4_8IOL:I.Data[86].0   // IO-Link Port 6 - Input data word 3 (INT bit0)
           TBEN_L4_8IOL:I.Data[86].1   // IO-Link Port 6 - Input data word 3 (INT bit1)
           TBEN_L4_8IOL:I.Data[86].10   // IO-Link Port 6 - Input data word 3 (INT bit10)
           TBEN_L4_8IOL:I.Data[86].11   // IO-Link Port 6 - Input data word 3 (INT bit11)
           TBEN_L4_8IOL:I.Data[86].12   // IO-Link Port 6 - Input data word 3 (INT bit12)
           TBEN_L4_8IOL:I.Data[86].13   // IO-Link Port 6 - Input data word 3 (INT bit13)
           TBEN_L4_8IOL:I.Data[86].14   // IO-Link Port 6 - Input data word 3 (INT bit14)
           TBEN_L4_8IOL:I.Data[86].15   // IO-Link Port 6 - Input data word 3 (INT bit15)
           TBEN_L4_8IOL:I.Data[86].2   // IO-Link Port 6 - Input data word 3 (INT bit2)
           TBEN_L4_8IOL:I.Data[86].3   // IO-Link Port 6 - Input data word 3 (INT bit3)
           TBEN_L4_8IOL:I.Data[86].4   // IO-Link Port 6 - Input data word 3 (INT bit4)
           TBEN_L4_8IOL:I.Data[86].5   // IO-Link Port 6 - Input data word 3 (INT bit5)
           TBEN_L4_8IOL:I.Data[86].6   // IO-Link Port 6 - Input data word 3 (INT bit6)
           TBEN_L4_8IOL:I.Data[86].7   // IO-Link Port 6 - Input data word 3 (INT bit7)
           TBEN_L4_8IOL:I.Data[86].8   // IO-Link Port 6 - Input data word 3 (INT bit8)
           TBEN_L4_8IOL:I.Data[86].9   // IO-Link Port 6 - Input data word 3 (INT bit9)
           TBEN_L4_8IOL:I.Data[87]   // IO-Link Port 6 - Input data word 4
           TBEN_L4_8IOL:I.Data[87].0   // IO-Link Port 6 - Input data word 4 (INT bit0)
           TBEN_L4_8IOL:I.Data[87].1   // IO-Link Port 6 - Input data word 4 (INT bit1)
           TBEN_L4_8IOL:I.Data[87].10   // IO-Link Port 6 - Input data word 4 (INT bit10)
           TBEN_L4_8IOL:I.Data[87].11   // IO-Link Port 6 - Input data word 4 (INT bit11)
           TBEN_L4_8IOL:I.Data[87].12   // IO-Link Port 6 - Input data word 4 (INT bit12)
           TBEN_L4_8IOL:I.Data[87].13   // IO-Link Port 6 - Input data word 4 (INT bit13)
           TBEN_L4_8IOL:I.Data[87].14   // IO-Link Port 6 - Input data word 4 (INT bit14)
           TBEN_L4_8IOL:I.Data[87].15   // IO-Link Port 6 - Input data word 4 (INT bit15)
           TBEN_L4_8IOL:I.Data[87].2   // IO-Link Port 6 - Input data word 4 (INT bit2)
           TBEN_L4_8IOL:I.Data[87].3   // IO-Link Port 6 - Input data word 4 (INT bit3)
           TBEN_L4_8IOL:I.Data[87].4   // IO-Link Port 6 - Input data word 4 (INT bit4)
           TBEN_L4_8IOL:I.Data[87].5   // IO-Link Port 6 - Input data word 4 (INT bit5)
           TBEN_L4_8IOL:I.Data[87].6   // IO-Link Port 6 - Input data word 4 (INT bit6)
           TBEN_L4_8IOL:I.Data[87].7   // IO-Link Port 6 - Input data word 4 (INT bit7)
           TBEN_L4_8IOL:I.Data[87].8   // IO-Link Port 6 - Input data word 4 (INT bit8)
           TBEN_L4_8IOL:I.Data[87].9   // IO-Link Port 6 - Input data word 4 (INT bit9)
           TBEN_L4_8IOL:I.Data[88]   // IO-Link Port 6 - Input data word 5
           TBEN_L4_8IOL:I.Data[88].0   // IO-Link Port 6 - Input data word 5 (INT bit0)
           TBEN_L4_8IOL:I.Data[88].1   // IO-Link Port 6 - Input data word 5 (INT bit1)
           TBEN_L4_8IOL:I.Data[88].10   // IO-Link Port 6 - Input data word 5 (INT bit10)
           TBEN_L4_8IOL:I.Data[88].11   // IO-Link Port 6 - Input data word 5 (INT bit11)
           TBEN_L4_8IOL:I.Data[88].12   // IO-Link Port 6 - Input data word 5 (INT bit12)
           TBEN_L4_8IOL:I.Data[88].13   // IO-Link Port 6 - Input data word 5 (INT bit13)
           TBEN_L4_8IOL:I.Data[88].14   // IO-Link Port 6 - Input data word 5 (INT bit14)
           TBEN_L4_8IOL:I.Data[88].15   // IO-Link Port 6 - Input data word 5 (INT bit15)
           TBEN_L4_8IOL:I.Data[88].2   // IO-Link Port 6 - Input data word 5 (INT bit2)
           TBEN_L4_8IOL:I.Data[88].3   // IO-Link Port 6 - Input data word 5 (INT bit3)
           TBEN_L4_8IOL:I.Data[88].4   // IO-Link Port 6 - Input data word 5 (INT bit4)
           TBEN_L4_8IOL:I.Data[88].5   // IO-Link Port 6 - Input data word 5 (INT bit5)
           TBEN_L4_8IOL:I.Data[88].6   // IO-Link Port 6 - Input data word 5 (INT bit6)
           TBEN_L4_8IOL:I.Data[88].7   // IO-Link Port 6 - Input data word 5 (INT bit7)
           TBEN_L4_8IOL:I.Data[88].8   // IO-Link Port 6 - Input data word 5 (INT bit8)
           TBEN_L4_8IOL:I.Data[88].9   // IO-Link Port 6 - Input data word 5 (INT bit9)
           TBEN_L4_8IOL:I.Data[89]   // IO-Link Port 6 - Input data word 6
           TBEN_L4_8IOL:I.Data[89].0   // IO-Link Port 6 - Input data word 6 (INT bit0)
           TBEN_L4_8IOL:I.Data[89].1   // IO-Link Port 6 - Input data word 6 (INT bit1)
           TBEN_L4_8IOL:I.Data[89].10   // IO-Link Port 6 - Input data word 6 (INT bit10)
           TBEN_L4_8IOL:I.Data[89].11   // IO-Link Port 6 - Input data word 6 (INT bit11)
           TBEN_L4_8IOL:I.Data[89].12   // IO-Link Port 6 - Input data word 6 (INT bit12)
           TBEN_L4_8IOL:I.Data[89].13   // IO-Link Port 6 - Input data word 6 (INT bit13)
           TBEN_L4_8IOL:I.Data[89].14   // IO-Link Port 6 - Input data word 6 (INT bit14)
           TBEN_L4_8IOL:I.Data[89].15   // IO-Link Port 6 - Input data word 6 (INT bit15)
           TBEN_L4_8IOL:I.Data[89].2   // IO-Link Port 6 - Input data word 6 (INT bit2)
           TBEN_L4_8IOL:I.Data[89].3   // IO-Link Port 6 - Input data word 6 (INT bit3)
           TBEN_L4_8IOL:I.Data[89].4   // IO-Link Port 6 - Input data word 6 (INT bit4)
           TBEN_L4_8IOL:I.Data[89].5   // IO-Link Port 6 - Input data word 6 (INT bit5)
           TBEN_L4_8IOL:I.Data[89].6   // IO-Link Port 6 - Input data word 6 (INT bit6)
           TBEN_L4_8IOL:I.Data[89].7   // IO-Link Port 6 - Input data word 6 (INT bit7)
           TBEN_L4_8IOL:I.Data[89].8   // IO-Link Port 6 - Input data word 6 (INT bit8)
           TBEN_L4_8IOL:I.Data[89].9   // IO-Link Port 6 - Input data word 6 (INT bit9)
           TBEN_L4_8IOL:I.Data[8]   // IO-Link Port 1 - Input data word 5
           TBEN_L4_8IOL:I.Data[8].0   // IO-Link Port 1 - Input data word 5 (INT bit0)
           TBEN_L4_8IOL:I.Data[8].1   // IO-Link Port 1 - Input data word 5 (INT bit1)
           TBEN_L4_8IOL:I.Data[8].10   // IO-Link Port 1 - Input data word 5 (INT bit10)
           TBEN_L4_8IOL:I.Data[8].11   // IO-Link Port 1 - Input data word 5 (INT bit11)
           TBEN_L4_8IOL:I.Data[8].12   // IO-Link Port 1 - Input data word 5 (INT bit12)
           TBEN_L4_8IOL:I.Data[8].13   // IO-Link Port 1 - Input data word 5 (INT bit13)
           TBEN_L4_8IOL:I.Data[8].14   // IO-Link Port 1 - Input data word 5 (INT bit14)
           TBEN_L4_8IOL:I.Data[8].15   // IO-Link Port 1 - Input data word 5 (INT bit15)
           TBEN_L4_8IOL:I.Data[8].2   // IO-Link Port 1 - Input data word 5 (INT bit2)
           TBEN_L4_8IOL:I.Data[8].3   // IO-Link Port 1 - Input data word 5 (INT bit3)
           TBEN_L4_8IOL:I.Data[8].4   // IO-Link Port 1 - Input data word 5 (INT bit4)
           TBEN_L4_8IOL:I.Data[8].5   // IO-Link Port 1 - Input data word 5 (INT bit5)
           TBEN_L4_8IOL:I.Data[8].6   // IO-Link Port 1 - Input data word 5 (INT bit6)
           TBEN_L4_8IOL:I.Data[8].7   // IO-Link Port 1 - Input data word 5 (INT bit7)
           TBEN_L4_8IOL:I.Data[8].8   // IO-Link Port 1 - Input data word 5 (INT bit8)
           TBEN_L4_8IOL:I.Data[8].9   // IO-Link Port 1 - Input data word 5 (INT bit9)
           TBEN_L4_8IOL:I.Data[90]   // IO-Link Port 6 - Input data word 7
           TBEN_L4_8IOL:I.Data[90].0   // IO-Link Port 6 - Input data word 7 (INT bit0)
           TBEN_L4_8IOL:I.Data[90].1   // IO-Link Port 6 - Input data word 7 (INT bit1)
           TBEN_L4_8IOL:I.Data[90].10   // IO-Link Port 6 - Input data word 7 (INT bit10)
           TBEN_L4_8IOL:I.Data[90].11   // IO-Link Port 6 - Input data word 7 (INT bit11)
           TBEN_L4_8IOL:I.Data[90].12   // IO-Link Port 6 - Input data word 7 (INT bit12)
           TBEN_L4_8IOL:I.Data[90].13   // IO-Link Port 6 - Input data word 7 (INT bit13)
           TBEN_L4_8IOL:I.Data[90].14   // IO-Link Port 6 - Input data word 7 (INT bit14)
           TBEN_L4_8IOL:I.Data[90].15   // IO-Link Port 6 - Input data word 7 (INT bit15)
           TBEN_L4_8IOL:I.Data[90].2   // IO-Link Port 6 - Input data word 7 (INT bit2)
           TBEN_L4_8IOL:I.Data[90].3   // IO-Link Port 6 - Input data word 7 (INT bit3)
           TBEN_L4_8IOL:I.Data[90].4   // IO-Link Port 6 - Input data word 7 (INT bit4)
           TBEN_L4_8IOL:I.Data[90].5   // IO-Link Port 6 - Input data word 7 (INT bit5)
           TBEN_L4_8IOL:I.Data[90].6   // IO-Link Port 6 - Input data word 7 (INT bit6)
           TBEN_L4_8IOL:I.Data[90].7   // IO-Link Port 6 - Input data word 7 (INT bit7)
           TBEN_L4_8IOL:I.Data[90].8   // IO-Link Port 6 - Input data word 7 (INT bit8)
           TBEN_L4_8IOL:I.Data[90].9   // IO-Link Port 6 - Input data word 7 (INT bit9)
           TBEN_L4_8IOL:I.Data[91]   // IO-Link Port 6 - Input data word 8
           TBEN_L4_8IOL:I.Data[91].0   // IO-Link Port 6 - Input data word 8 (INT bit0)
           TBEN_L4_8IOL:I.Data[91].1   // IO-Link Port 6 - Input data word 8 (INT bit1)
           TBEN_L4_8IOL:I.Data[91].10   // IO-Link Port 6 - Input data word 8 (INT bit10)
           TBEN_L4_8IOL:I.Data[91].11   // IO-Link Port 6 - Input data word 8 (INT bit11)
           TBEN_L4_8IOL:I.Data[91].12   // IO-Link Port 6 - Input data word 8 (INT bit12)
           TBEN_L4_8IOL:I.Data[91].13   // IO-Link Port 6 - Input data word 8 (INT bit13)
           TBEN_L4_8IOL:I.Data[91].14   // IO-Link Port 6 - Input data word 8 (INT bit14)
           TBEN_L4_8IOL:I.Data[91].15   // IO-Link Port 6 - Input data word 8 (INT bit15)
           TBEN_L4_8IOL:I.Data[91].2   // IO-Link Port 6 - Input data word 8 (INT bit2)
           TBEN_L4_8IOL:I.Data[91].3   // IO-Link Port 6 - Input data word 8 (INT bit3)
           TBEN_L4_8IOL:I.Data[91].4   // IO-Link Port 6 - Input data word 8 (INT bit4)
           TBEN_L4_8IOL:I.Data[91].5   // IO-Link Port 6 - Input data word 8 (INT bit5)
           TBEN_L4_8IOL:I.Data[91].6   // IO-Link Port 6 - Input data word 8 (INT bit6)
           TBEN_L4_8IOL:I.Data[91].7   // IO-Link Port 6 - Input data word 8 (INT bit7)
           TBEN_L4_8IOL:I.Data[91].8   // IO-Link Port 6 - Input data word 8 (INT bit8)
           TBEN_L4_8IOL:I.Data[91].9   // IO-Link Port 6 - Input data word 8 (INT bit9)
           TBEN_L4_8IOL:I.Data[92]   // IO-Link Port 6 - Input data word 9
           TBEN_L4_8IOL:I.Data[92].0   // IO-Link Port 6 - Input data word 9 (INT bit0)
           TBEN_L4_8IOL:I.Data[92].1   // IO-Link Port 6 - Input data word 9 (INT bit1)
           TBEN_L4_8IOL:I.Data[92].10   // IO-Link Port 6 - Input data word 9 (INT bit10)
           TBEN_L4_8IOL:I.Data[92].11   // IO-Link Port 6 - Input data word 9 (INT bit11)
           TBEN_L4_8IOL:I.Data[92].12   // IO-Link Port 6 - Input data word 9 (INT bit12)
           TBEN_L4_8IOL:I.Data[92].13   // IO-Link Port 6 - Input data word 9 (INT bit13)
           TBEN_L4_8IOL:I.Data[92].14   // IO-Link Port 6 - Input data word 9 (INT bit14)
           TBEN_L4_8IOL:I.Data[92].15   // IO-Link Port 6 - Input data word 9 (INT bit15)
           TBEN_L4_8IOL:I.Data[92].2   // IO-Link Port 6 - Input data word 9 (INT bit2)
           TBEN_L4_8IOL:I.Data[92].3   // IO-Link Port 6 - Input data word 9 (INT bit3)
           TBEN_L4_8IOL:I.Data[92].4   // IO-Link Port 6 - Input data word 9 (INT bit4)
           TBEN_L4_8IOL:I.Data[92].5   // IO-Link Port 6 - Input data word 9 (INT bit5)
           TBEN_L4_8IOL:I.Data[92].6   // IO-Link Port 6 - Input data word 9 (INT bit6)
           TBEN_L4_8IOL:I.Data[92].7   // IO-Link Port 6 - Input data word 9 (INT bit7)
           TBEN_L4_8IOL:I.Data[92].8   // IO-Link Port 6 - Input data word 9 (INT bit8)
           TBEN_L4_8IOL:I.Data[92].9   // IO-Link Port 6 - Input data word 9 (INT bit9)
           TBEN_L4_8IOL:I.Data[93]   // IO-Link Port 6 - Input data word 10
           TBEN_L4_8IOL:I.Data[93].0   // IO-Link Port 6 - Input data word 10 (INT bit0)
           TBEN_L4_8IOL:I.Data[93].1   // IO-Link Port 6 - Input data word 10 (INT bit1)
           TBEN_L4_8IOL:I.Data[93].10   // IO-Link Port 6 - Input data word 10 (INT bit10)
           TBEN_L4_8IOL:I.Data[93].11   // IO-Link Port 6 - Input data word 10 (INT bit11)
           TBEN_L4_8IOL:I.Data[93].12   // IO-Link Port 6 - Input data word 10 (INT bit12)
           TBEN_L4_8IOL:I.Data[93].13   // IO-Link Port 6 - Input data word 10 (INT bit13)
           TBEN_L4_8IOL:I.Data[93].14   // IO-Link Port 6 - Input data word 10 (INT bit14)
           TBEN_L4_8IOL:I.Data[93].15   // IO-Link Port 6 - Input data word 10 (INT bit15)
           TBEN_L4_8IOL:I.Data[93].2   // IO-Link Port 6 - Input data word 10 (INT bit2)
           TBEN_L4_8IOL:I.Data[93].3   // IO-Link Port 6 - Input data word 10 (INT bit3)
           TBEN_L4_8IOL:I.Data[93].4   // IO-Link Port 6 - Input data word 10 (INT bit4)
           TBEN_L4_8IOL:I.Data[93].5   // IO-Link Port 6 - Input data word 10 (INT bit5)
           TBEN_L4_8IOL:I.Data[93].6   // IO-Link Port 6 - Input data word 10 (INT bit6)
           TBEN_L4_8IOL:I.Data[93].7   // IO-Link Port 6 - Input data word 10 (INT bit7)
           TBEN_L4_8IOL:I.Data[93].8   // IO-Link Port 6 - Input data word 10 (INT bit8)
           TBEN_L4_8IOL:I.Data[93].9   // IO-Link Port 6 - Input data word 10 (INT bit9)
           TBEN_L4_8IOL:I.Data[94]   // IO-Link Port 6 - Input data word 11
           TBEN_L4_8IOL:I.Data[94].0   // IO-Link Port 6 - Input data word 11 (INT bit0)
           TBEN_L4_8IOL:I.Data[94].1   // IO-Link Port 6 - Input data word 11 (INT bit1)
           TBEN_L4_8IOL:I.Data[94].10   // IO-Link Port 6 - Input data word 11 (INT bit10)
           TBEN_L4_8IOL:I.Data[94].11   // IO-Link Port 6 - Input data word 11 (INT bit11)
           TBEN_L4_8IOL:I.Data[94].12   // IO-Link Port 6 - Input data word 11 (INT bit12)
           TBEN_L4_8IOL:I.Data[94].13   // IO-Link Port 6 - Input data word 11 (INT bit13)
           TBEN_L4_8IOL:I.Data[94].14   // IO-Link Port 6 - Input data word 11 (INT bit14)
           TBEN_L4_8IOL:I.Data[94].15   // IO-Link Port 6 - Input data word 11 (INT bit15)
           TBEN_L4_8IOL:I.Data[94].2   // IO-Link Port 6 - Input data word 11 (INT bit2)
           TBEN_L4_8IOL:I.Data[94].3   // IO-Link Port 6 - Input data word 11 (INT bit3)
           TBEN_L4_8IOL:I.Data[94].4   // IO-Link Port 6 - Input data word 11 (INT bit4)
           TBEN_L4_8IOL:I.Data[94].5   // IO-Link Port 6 - Input data word 11 (INT bit5)
           TBEN_L4_8IOL:I.Data[94].6   // IO-Link Port 6 - Input data word 11 (INT bit6)
           TBEN_L4_8IOL:I.Data[94].7   // IO-Link Port 6 - Input data word 11 (INT bit7)
           TBEN_L4_8IOL:I.Data[94].8   // IO-Link Port 6 - Input data word 11 (INT bit8)
           TBEN_L4_8IOL:I.Data[94].9   // IO-Link Port 6 - Input data word 11 (INT bit9)
           TBEN_L4_8IOL:I.Data[95]   // IO-Link Port 6 - Input data word 12
           TBEN_L4_8IOL:I.Data[95].0   // IO-Link Port 6 - Input data word 12 (INT bit0)
           TBEN_L4_8IOL:I.Data[95].1   // IO-Link Port 6 - Input data word 12 (INT bit1)
           TBEN_L4_8IOL:I.Data[95].10   // IO-Link Port 6 - Input data word 12 (INT bit10)
           TBEN_L4_8IOL:I.Data[95].11   // IO-Link Port 6 - Input data word 12 (INT bit11)
           TBEN_L4_8IOL:I.Data[95].12   // IO-Link Port 6 - Input data word 12 (INT bit12)
           TBEN_L4_8IOL:I.Data[95].13   // IO-Link Port 6 - Input data word 12 (INT bit13)
           TBEN_L4_8IOL:I.Data[95].14   // IO-Link Port 6 - Input data word 12 (INT bit14)
           TBEN_L4_8IOL:I.Data[95].15   // IO-Link Port 6 - Input data word 12 (INT bit15)
           TBEN_L4_8IOL:I.Data[95].2   // IO-Link Port 6 - Input data word 12 (INT bit2)
           TBEN_L4_8IOL:I.Data[95].3   // IO-Link Port 6 - Input data word 12 (INT bit3)
           TBEN_L4_8IOL:I.Data[95].4   // IO-Link Port 6 - Input data word 12 (INT bit4)
           TBEN_L4_8IOL:I.Data[95].5   // IO-Link Port 6 - Input data word 12 (INT bit5)
           TBEN_L4_8IOL:I.Data[95].6   // IO-Link Port 6 - Input data word 12 (INT bit6)
           TBEN_L4_8IOL:I.Data[95].7   // IO-Link Port 6 - Input data word 12 (INT bit7)
           TBEN_L4_8IOL:I.Data[95].8   // IO-Link Port 6 - Input data word 12 (INT bit8)
           TBEN_L4_8IOL:I.Data[95].9   // IO-Link Port 6 - Input data word 12 (INT bit9)
           TBEN_L4_8IOL:I.Data[96]   // IO-Link Port 6 - Input data word 13
           TBEN_L4_8IOL:I.Data[96].0   // IO-Link Port 6 - Input data word 13 (INT bit0)
           TBEN_L4_8IOL:I.Data[96].1   // IO-Link Port 6 - Input data word 13 (INT bit1)
           TBEN_L4_8IOL:I.Data[96].10   // IO-Link Port 6 - Input data word 13 (INT bit10)
           TBEN_L4_8IOL:I.Data[96].11   // IO-Link Port 6 - Input data word 13 (INT bit11)
           TBEN_L4_8IOL:I.Data[96].12   // IO-Link Port 6 - Input data word 13 (INT bit12)
           TBEN_L4_8IOL:I.Data[96].13   // IO-Link Port 6 - Input data word 13 (INT bit13)
           TBEN_L4_8IOL:I.Data[96].14   // IO-Link Port 6 - Input data word 13 (INT bit14)
           TBEN_L4_8IOL:I.Data[96].15   // IO-Link Port 6 - Input data word 13 (INT bit15)
           TBEN_L4_8IOL:I.Data[96].2   // IO-Link Port 6 - Input data word 13 (INT bit2)
           TBEN_L4_8IOL:I.Data[96].3   // IO-Link Port 6 - Input data word 13 (INT bit3)
           TBEN_L4_8IOL:I.Data[96].4   // IO-Link Port 6 - Input data word 13 (INT bit4)
           TBEN_L4_8IOL:I.Data[96].5   // IO-Link Port 6 - Input data word 13 (INT bit5)
           TBEN_L4_8IOL:I.Data[96].6   // IO-Link Port 6 - Input data word 13 (INT bit6)
           TBEN_L4_8IOL:I.Data[96].7   // IO-Link Port 6 - Input data word 13 (INT bit7)
           TBEN_L4_8IOL:I.Data[96].8   // IO-Link Port 6 - Input data word 13 (INT bit8)
           TBEN_L4_8IOL:I.Data[96].9   // IO-Link Port 6 - Input data word 13 (INT bit9)
           TBEN_L4_8IOL:I.Data[97]   // IO-Link Port 6 - Input data word 14
           TBEN_L4_8IOL:I.Data[97].0   // IO-Link Port 6 - Input data word 14 (INT bit0)
           TBEN_L4_8IOL:I.Data[97].1   // IO-Link Port 6 - Input data word 14 (INT bit1)
           TBEN_L4_8IOL:I.Data[97].10   // IO-Link Port 6 - Input data word 14 (INT bit10)
           TBEN_L4_8IOL:I.Data[97].11   // IO-Link Port 6 - Input data word 14 (INT bit11)
           TBEN_L4_8IOL:I.Data[97].12   // IO-Link Port 6 - Input data word 14 (INT bit12)
           TBEN_L4_8IOL:I.Data[97].13   // IO-Link Port 6 - Input data word 14 (INT bit13)
           TBEN_L4_8IOL:I.Data[97].14   // IO-Link Port 6 - Input data word 14 (INT bit14)
           TBEN_L4_8IOL:I.Data[97].15   // IO-Link Port 6 - Input data word 14 (INT bit15)
           TBEN_L4_8IOL:I.Data[97].2   // IO-Link Port 6 - Input data word 14 (INT bit2)
           TBEN_L4_8IOL:I.Data[97].3   // IO-Link Port 6 - Input data word 14 (INT bit3)
           TBEN_L4_8IOL:I.Data[97].4   // IO-Link Port 6 - Input data word 14 (INT bit4)
           TBEN_L4_8IOL:I.Data[97].5   // IO-Link Port 6 - Input data word 14 (INT bit5)
           TBEN_L4_8IOL:I.Data[97].6   // IO-Link Port 6 - Input data word 14 (INT bit6)
           TBEN_L4_8IOL:I.Data[97].7   // IO-Link Port 6 - Input data word 14 (INT bit7)
           TBEN_L4_8IOL:I.Data[97].8   // IO-Link Port 6 - Input data word 14 (INT bit8)
           TBEN_L4_8IOL:I.Data[97].9   // IO-Link Port 6 - Input data word 14 (INT bit9)
           TBEN_L4_8IOL:I.Data[98]   // IO-Link Port 6 - Input data word 15
           TBEN_L4_8IOL:I.Data[98].0   // IO-Link Port 6 - Input data word 15 (INT bit0)
           TBEN_L4_8IOL:I.Data[98].1   // IO-Link Port 6 - Input data word 15 (INT bit1)
           TBEN_L4_8IOL:I.Data[98].10   // IO-Link Port 6 - Input data word 15 (INT bit10)
           TBEN_L4_8IOL:I.Data[98].11   // IO-Link Port 6 - Input data word 15 (INT bit11)
           TBEN_L4_8IOL:I.Data[98].12   // IO-Link Port 6 - Input data word 15 (INT bit12)
           TBEN_L4_8IOL:I.Data[98].13   // IO-Link Port 6 - Input data word 15 (INT bit13)
           TBEN_L4_8IOL:I.Data[98].14   // IO-Link Port 6 - Input data word 15 (INT bit14)
           TBEN_L4_8IOL:I.Data[98].15   // IO-Link Port 6 - Input data word 15 (INT bit15)
           TBEN_L4_8IOL:I.Data[98].2   // IO-Link Port 6 - Input data word 15 (INT bit2)
           TBEN_L4_8IOL:I.Data[98].3   // IO-Link Port 6 - Input data word 15 (INT bit3)
           TBEN_L4_8IOL:I.Data[98].4   // IO-Link Port 6 - Input data word 15 (INT bit4)
           TBEN_L4_8IOL:I.Data[98].5   // IO-Link Port 6 - Input data word 15 (INT bit5)
           TBEN_L4_8IOL:I.Data[98].6   // IO-Link Port 6 - Input data word 15 (INT bit6)
           TBEN_L4_8IOL:I.Data[98].7   // IO-Link Port 6 - Input data word 15 (INT bit7)
           TBEN_L4_8IOL:I.Data[98].8   // IO-Link Port 6 - Input data word 15 (INT bit8)
           TBEN_L4_8IOL:I.Data[98].9   // IO-Link Port 6 - Input data word 15 (INT bit9)
           TBEN_L4_8IOL:I.Data[99]   // IO-Link Port 7 - Input data word 0
           TBEN_L4_8IOL:I.Data[99].0   // IO-Link Port 7 - Input data word 0 (INT bit0)
           TBEN_L4_8IOL:I.Data[99].1   // IO-Link Port 7 - Input data word 0 (INT bit1)
           TBEN_L4_8IOL:I.Data[99].10   // IO-Link Port 7 - Input data word 0 (INT bit10)
           TBEN_L4_8IOL:I.Data[99].11   // IO-Link Port 7 - Input data word 0 (INT bit11)
           TBEN_L4_8IOL:I.Data[99].12   // IO-Link Port 7 - Input data word 0 (INT bit12)
           TBEN_L4_8IOL:I.Data[99].13   // IO-Link Port 7 - Input data word 0 (INT bit13)
           TBEN_L4_8IOL:I.Data[99].14   // IO-Link Port 7 - Input data word 0 (INT bit14)
           TBEN_L4_8IOL:I.Data[99].15   // IO-Link Port 7 - Input data word 0 (INT bit15)
           TBEN_L4_8IOL:I.Data[99].2   // IO-Link Port 7 - Input data word 0 (INT bit2)
           TBEN_L4_8IOL:I.Data[99].3   // IO-Link Port 7 - Input data word 0 (INT bit3)
           TBEN_L4_8IOL:I.Data[99].4   // IO-Link Port 7 - Input data word 0 (INT bit4)
           TBEN_L4_8IOL:I.Data[99].5   // IO-Link Port 7 - Input data word 0 (INT bit5)
           TBEN_L4_8IOL:I.Data[99].6   // IO-Link Port 7 - Input data word 0 (INT bit6)
           TBEN_L4_8IOL:I.Data[99].7   // IO-Link Port 7 - Input data word 0 (INT bit7)
           TBEN_L4_8IOL:I.Data[99].8   // IO-Link Port 7 - Input data word 0 (INT bit8)
           TBEN_L4_8IOL:I.Data[99].9   // IO-Link Port 7 - Input data word 0 (INT bit9)
           TBEN_L4_8IOL:I.Data[9]   // IO-Link Port 1 - Input data word 6
           TBEN_L4_8IOL:I.Data[9].0   // IO-Link Port 1 - Input data word 6 (INT bit0)
           TBEN_L4_8IOL:I.Data[9].1   // IO-Link Port 1 - Input data word 6 (INT bit1)
           TBEN_L4_8IOL:I.Data[9].10   // IO-Link Port 1 - Input data word 6 (INT bit10)
           TBEN_L4_8IOL:I.Data[9].11   // IO-Link Port 1 - Input data word 6 (INT bit11)
           TBEN_L4_8IOL:I.Data[9].12   // IO-Link Port 1 - Input data word 6 (INT bit12)
           TBEN_L4_8IOL:I.Data[9].13   // IO-Link Port 1 - Input data word 6 (INT bit13)
           TBEN_L4_8IOL:I.Data[9].14   // IO-Link Port 1 - Input data word 6 (INT bit14)
           TBEN_L4_8IOL:I.Data[9].15   // IO-Link Port 1 - Input data word 6 (INT bit15)
           TBEN_L4_8IOL:I.Data[9].2   // IO-Link Port 1 - Input data word 6 (INT bit2)
           TBEN_L4_8IOL:I.Data[9].3   // IO-Link Port 1 - Input data word 6 (INT bit3)
           TBEN_L4_8IOL:I.Data[9].4   // IO-Link Port 1 - Input data word 6 (INT bit4)
           TBEN_L4_8IOL:I.Data[9].5   // IO-Link Port 1 - Input data word 6 (INT bit5)
           TBEN_L4_8IOL:I.Data[9].6   // IO-Link Port 1 - Input data word 6 (INT bit6)
           TBEN_L4_8IOL:I.Data[9].7   // IO-Link Port 1 - Input data word 6 (INT bit7)
           TBEN_L4_8IOL:I.Data[9].8   // IO-Link Port 1 - Input data word 6 (INT bit8)
           TBEN_L4_8IOL:I.Data[9].9   // IO-Link Port 1 - Input data word 6 (INT bit9)
           TBEN_L4_8IOL:O.Data[0]   // Station Control Word
           TBEN_L4_8IOL:O.Data[100]   // IO-Link Port 7 - Output data word 2
           TBEN_L4_8IOL:O.Data[100].0   // IO-Link Port 7 - Output data word 2 (INT bit0)
           TBEN_L4_8IOL:O.Data[100].1   // IO-Link Port 7 - Output data word 2 (INT bit1)
           TBEN_L4_8IOL:O.Data[100].10   // IO-Link Port 7 - Output data word 2 (INT bit10)
           TBEN_L4_8IOL:O.Data[100].11   // IO-Link Port 7 - Output data word 2 (INT bit11)
           TBEN_L4_8IOL:O.Data[100].12   // IO-Link Port 7 - Output data word 2 (INT bit12)
           TBEN_L4_8IOL:O.Data[100].13   // IO-Link Port 7 - Output data word 2 (INT bit13)
           TBEN_L4_8IOL:O.Data[100].14   // IO-Link Port 7 - Output data word 2 (INT bit14)
           TBEN_L4_8IOL:O.Data[100].15   // IO-Link Port 7 - Output data word 2 (INT bit15)
           TBEN_L4_8IOL:O.Data[100].2   // IO-Link Port 7 - Output data word 2 (INT bit2)
           TBEN_L4_8IOL:O.Data[100].3   // IO-Link Port 7 - Output data word 2 (INT bit3)
           TBEN_L4_8IOL:O.Data[100].4   // IO-Link Port 7 - Output data word 2 (INT bit4)
           TBEN_L4_8IOL:O.Data[100].5   // IO-Link Port 7 - Output data word 2 (INT bit5)
           TBEN_L4_8IOL:O.Data[100].6   // IO-Link Port 7 - Output data word 2 (INT bit6)
           TBEN_L4_8IOL:O.Data[100].7   // IO-Link Port 7 - Output data word 2 (INT bit7)
           TBEN_L4_8IOL:O.Data[100].8   // IO-Link Port 7 - Output data word 2 (INT bit8)
           TBEN_L4_8IOL:O.Data[100].9   // IO-Link Port 7 - Output data word 2 (INT bit9)
           TBEN_L4_8IOL:O.Data[101]   // IO-Link Port 7 - Output data word 3
           TBEN_L4_8IOL:O.Data[101].0   // IO-Link Port 7 - Output data word 3 (INT bit0)
           TBEN_L4_8IOL:O.Data[101].1   // IO-Link Port 7 - Output data word 3 (INT bit1)
           TBEN_L4_8IOL:O.Data[101].10   // IO-Link Port 7 - Output data word 3 (INT bit10)
           TBEN_L4_8IOL:O.Data[101].11   // IO-Link Port 7 - Output data word 3 (INT bit11)
           TBEN_L4_8IOL:O.Data[101].12   // IO-Link Port 7 - Output data word 3 (INT bit12)
           TBEN_L4_8IOL:O.Data[101].13   // IO-Link Port 7 - Output data word 3 (INT bit13)
           TBEN_L4_8IOL:O.Data[101].14   // IO-Link Port 7 - Output data word 3 (INT bit14)
           TBEN_L4_8IOL:O.Data[101].15   // IO-Link Port 7 - Output data word 3 (INT bit15)
           TBEN_L4_8IOL:O.Data[101].2   // IO-Link Port 7 - Output data word 3 (INT bit2)
           TBEN_L4_8IOL:O.Data[101].3   // IO-Link Port 7 - Output data word 3 (INT bit3)
           TBEN_L4_8IOL:O.Data[101].4   // IO-Link Port 7 - Output data word 3 (INT bit4)
           TBEN_L4_8IOL:O.Data[101].5   // IO-Link Port 7 - Output data word 3 (INT bit5)
           TBEN_L4_8IOL:O.Data[101].6   // IO-Link Port 7 - Output data word 3 (INT bit6)
           TBEN_L4_8IOL:O.Data[101].7   // IO-Link Port 7 - Output data word 3 (INT bit7)
           TBEN_L4_8IOL:O.Data[101].8   // IO-Link Port 7 - Output data word 3 (INT bit8)
           TBEN_L4_8IOL:O.Data[101].9   // IO-Link Port 7 - Output data word 3 (INT bit9)
           TBEN_L4_8IOL:O.Data[102]   // IO-Link Port 7 - Output data word 4
           TBEN_L4_8IOL:O.Data[102].0   // IO-Link Port 7 - Output data word 4 (INT bit0)
           TBEN_L4_8IOL:O.Data[102].1   // IO-Link Port 7 - Output data word 4 (INT bit1)
           TBEN_L4_8IOL:O.Data[102].10   // IO-Link Port 7 - Output data word 4 (INT bit10)
           TBEN_L4_8IOL:O.Data[102].11   // IO-Link Port 7 - Output data word 4 (INT bit11)
           TBEN_L4_8IOL:O.Data[102].12   // IO-Link Port 7 - Output data word 4 (INT bit12)
           TBEN_L4_8IOL:O.Data[102].13   // IO-Link Port 7 - Output data word 4 (INT bit13)
           TBEN_L4_8IOL:O.Data[102].14   // IO-Link Port 7 - Output data word 4 (INT bit14)
           TBEN_L4_8IOL:O.Data[102].15   // IO-Link Port 7 - Output data word 4 (INT bit15)
           TBEN_L4_8IOL:O.Data[102].2   // IO-Link Port 7 - Output data word 4 (INT bit2)
           TBEN_L4_8IOL:O.Data[102].3   // IO-Link Port 7 - Output data word 4 (INT bit3)
           TBEN_L4_8IOL:O.Data[102].4   // IO-Link Port 7 - Output data word 4 (INT bit4)
           TBEN_L4_8IOL:O.Data[102].5   // IO-Link Port 7 - Output data word 4 (INT bit5)
           TBEN_L4_8IOL:O.Data[102].6   // IO-Link Port 7 - Output data word 4 (INT bit6)
           TBEN_L4_8IOL:O.Data[102].7   // IO-Link Port 7 - Output data word 4 (INT bit7)
           TBEN_L4_8IOL:O.Data[102].8   // IO-Link Port 7 - Output data word 4 (INT bit8)
           TBEN_L4_8IOL:O.Data[102].9   // IO-Link Port 7 - Output data word 4 (INT bit9)
           TBEN_L4_8IOL:O.Data[103]   // IO-Link Port 7 - Output data word 5
           TBEN_L4_8IOL:O.Data[103].0   // IO-Link Port 7 - Output data word 5 (INT bit0)
           TBEN_L4_8IOL:O.Data[103].1   // IO-Link Port 7 - Output data word 5 (INT bit1)
           TBEN_L4_8IOL:O.Data[103].10   // IO-Link Port 7 - Output data word 5 (INT bit10)
           TBEN_L4_8IOL:O.Data[103].11   // IO-Link Port 7 - Output data word 5 (INT bit11)
           TBEN_L4_8IOL:O.Data[103].12   // IO-Link Port 7 - Output data word 5 (INT bit12)
           TBEN_L4_8IOL:O.Data[103].13   // IO-Link Port 7 - Output data word 5 (INT bit13)
           TBEN_L4_8IOL:O.Data[103].14   // IO-Link Port 7 - Output data word 5 (INT bit14)
           TBEN_L4_8IOL:O.Data[103].15   // IO-Link Port 7 - Output data word 5 (INT bit15)
           TBEN_L4_8IOL:O.Data[103].2   // IO-Link Port 7 - Output data word 5 (INT bit2)
           TBEN_L4_8IOL:O.Data[103].3   // IO-Link Port 7 - Output data word 5 (INT bit3)
           TBEN_L4_8IOL:O.Data[103].4   // IO-Link Port 7 - Output data word 5 (INT bit4)
           TBEN_L4_8IOL:O.Data[103].5   // IO-Link Port 7 - Output data word 5 (INT bit5)
           TBEN_L4_8IOL:O.Data[103].6   // IO-Link Port 7 - Output data word 5 (INT bit6)
           TBEN_L4_8IOL:O.Data[103].7   // IO-Link Port 7 - Output data word 5 (INT bit7)
           TBEN_L4_8IOL:O.Data[103].8   // IO-Link Port 7 - Output data word 5 (INT bit8)
           TBEN_L4_8IOL:O.Data[103].9   // IO-Link Port 7 - Output data word 5 (INT bit9)
           TBEN_L4_8IOL:O.Data[104]   // IO-Link Port 7 - Output data word 6
           TBEN_L4_8IOL:O.Data[104].0   // IO-Link Port 7 - Output data word 6 (INT bit0)
           TBEN_L4_8IOL:O.Data[104].1   // IO-Link Port 7 - Output data word 6 (INT bit1)
           TBEN_L4_8IOL:O.Data[104].10   // IO-Link Port 7 - Output data word 6 (INT bit10)
           TBEN_L4_8IOL:O.Data[104].11   // IO-Link Port 7 - Output data word 6 (INT bit11)
           TBEN_L4_8IOL:O.Data[104].12   // IO-Link Port 7 - Output data word 6 (INT bit12)
           TBEN_L4_8IOL:O.Data[104].13   // IO-Link Port 7 - Output data word 6 (INT bit13)
           TBEN_L4_8IOL:O.Data[104].14   // IO-Link Port 7 - Output data word 6 (INT bit14)
           TBEN_L4_8IOL:O.Data[104].15   // IO-Link Port 7 - Output data word 6 (INT bit15)
           TBEN_L4_8IOL:O.Data[104].2   // IO-Link Port 7 - Output data word 6 (INT bit2)
           TBEN_L4_8IOL:O.Data[104].3   // IO-Link Port 7 - Output data word 6 (INT bit3)
           TBEN_L4_8IOL:O.Data[104].4   // IO-Link Port 7 - Output data word 6 (INT bit4)
           TBEN_L4_8IOL:O.Data[104].5   // IO-Link Port 7 - Output data word 6 (INT bit5)
           TBEN_L4_8IOL:O.Data[104].6   // IO-Link Port 7 - Output data word 6 (INT bit6)
           TBEN_L4_8IOL:O.Data[104].7   // IO-Link Port 7 - Output data word 6 (INT bit7)
           TBEN_L4_8IOL:O.Data[104].8   // IO-Link Port 7 - Output data word 6 (INT bit8)
           TBEN_L4_8IOL:O.Data[104].9   // IO-Link Port 7 - Output data word 6 (INT bit9)
           TBEN_L4_8IOL:O.Data[105]   // IO-Link Port 7 - Output data word 7
           TBEN_L4_8IOL:O.Data[105].0   // IO-Link Port 7 - Output data word 7 (INT bit0)
           TBEN_L4_8IOL:O.Data[105].1   // IO-Link Port 7 - Output data word 7 (INT bit1)
           TBEN_L4_8IOL:O.Data[105].10   // IO-Link Port 7 - Output data word 7 (INT bit10)
           TBEN_L4_8IOL:O.Data[105].11   // IO-Link Port 7 - Output data word 7 (INT bit11)
           TBEN_L4_8IOL:O.Data[105].12   // IO-Link Port 7 - Output data word 7 (INT bit12)
           TBEN_L4_8IOL:O.Data[105].13   // IO-Link Port 7 - Output data word 7 (INT bit13)
           TBEN_L4_8IOL:O.Data[105].14   // IO-Link Port 7 - Output data word 7 (INT bit14)
           TBEN_L4_8IOL:O.Data[105].15   // IO-Link Port 7 - Output data word 7 (INT bit15)
           TBEN_L4_8IOL:O.Data[105].2   // IO-Link Port 7 - Output data word 7 (INT bit2)
           TBEN_L4_8IOL:O.Data[105].3   // IO-Link Port 7 - Output data word 7 (INT bit3)
           TBEN_L4_8IOL:O.Data[105].4   // IO-Link Port 7 - Output data word 7 (INT bit4)
           TBEN_L4_8IOL:O.Data[105].5   // IO-Link Port 7 - Output data word 7 (INT bit5)
           TBEN_L4_8IOL:O.Data[105].6   // IO-Link Port 7 - Output data word 7 (INT bit6)
           TBEN_L4_8IOL:O.Data[105].7   // IO-Link Port 7 - Output data word 7 (INT bit7)
           TBEN_L4_8IOL:O.Data[105].8   // IO-Link Port 7 - Output data word 7 (INT bit8)
           TBEN_L4_8IOL:O.Data[105].9   // IO-Link Port 7 - Output data word 7 (INT bit9)
           TBEN_L4_8IOL:O.Data[106]   // IO-Link Port 7 - Output data word 8
           TBEN_L4_8IOL:O.Data[106].0   // IO-Link Port 7 - Output data word 8 (INT bit0)
           TBEN_L4_8IOL:O.Data[106].1   // IO-Link Port 7 - Output data word 8 (INT bit1)
           TBEN_L4_8IOL:O.Data[106].10   // IO-Link Port 7 - Output data word 8 (INT bit10)
           TBEN_L4_8IOL:O.Data[106].11   // IO-Link Port 7 - Output data word 8 (INT bit11)
           TBEN_L4_8IOL:O.Data[106].12   // IO-Link Port 7 - Output data word 8 (INT bit12)
           TBEN_L4_8IOL:O.Data[106].13   // IO-Link Port 7 - Output data word 8 (INT bit13)
           TBEN_L4_8IOL:O.Data[106].14   // IO-Link Port 7 - Output data word 8 (INT bit14)
           TBEN_L4_8IOL:O.Data[106].15   // IO-Link Port 7 - Output data word 8 (INT bit15)
           TBEN_L4_8IOL:O.Data[106].2   // IO-Link Port 7 - Output data word 8 (INT bit2)
           TBEN_L4_8IOL:O.Data[106].3   // IO-Link Port 7 - Output data word 8 (INT bit3)
           TBEN_L4_8IOL:O.Data[106].4   // IO-Link Port 7 - Output data word 8 (INT bit4)
           TBEN_L4_8IOL:O.Data[106].5   // IO-Link Port 7 - Output data word 8 (INT bit5)
           TBEN_L4_8IOL:O.Data[106].6   // IO-Link Port 7 - Output data word 8 (INT bit6)
           TBEN_L4_8IOL:O.Data[106].7   // IO-Link Port 7 - Output data word 8 (INT bit7)
           TBEN_L4_8IOL:O.Data[106].8   // IO-Link Port 7 - Output data word 8 (INT bit8)
           TBEN_L4_8IOL:O.Data[106].9   // IO-Link Port 7 - Output data word 8 (INT bit9)
           TBEN_L4_8IOL:O.Data[107]   // IO-Link Port 7 - Output data word 9
           TBEN_L4_8IOL:O.Data[107].0   // IO-Link Port 7 - Output data word 9 (INT bit0)
           TBEN_L4_8IOL:O.Data[107].1   // IO-Link Port 7 - Output data word 9 (INT bit1)
           TBEN_L4_8IOL:O.Data[107].10   // IO-Link Port 7 - Output data word 9 (INT bit10)
           TBEN_L4_8IOL:O.Data[107].11   // IO-Link Port 7 - Output data word 9 (INT bit11)
           TBEN_L4_8IOL:O.Data[107].12   // IO-Link Port 7 - Output data word 9 (INT bit12)
           TBEN_L4_8IOL:O.Data[107].13   // IO-Link Port 7 - Output data word 9 (INT bit13)
           TBEN_L4_8IOL:O.Data[107].14   // IO-Link Port 7 - Output data word 9 (INT bit14)
           TBEN_L4_8IOL:O.Data[107].15   // IO-Link Port 7 - Output data word 9 (INT bit15)
           TBEN_L4_8IOL:O.Data[107].2   // IO-Link Port 7 - Output data word 9 (INT bit2)
           TBEN_L4_8IOL:O.Data[107].3   // IO-Link Port 7 - Output data word 9 (INT bit3)
           TBEN_L4_8IOL:O.Data[107].4   // IO-Link Port 7 - Output data word 9 (INT bit4)
           TBEN_L4_8IOL:O.Data[107].5   // IO-Link Port 7 - Output data word 9 (INT bit5)
           TBEN_L4_8IOL:O.Data[107].6   // IO-Link Port 7 - Output data word 9 (INT bit6)
           TBEN_L4_8IOL:O.Data[107].7   // IO-Link Port 7 - Output data word 9 (INT bit7)
           TBEN_L4_8IOL:O.Data[107].8   // IO-Link Port 7 - Output data word 9 (INT bit8)
           TBEN_L4_8IOL:O.Data[107].9   // IO-Link Port 7 - Output data word 9 (INT bit9)
           TBEN_L4_8IOL:O.Data[108]   // IO-Link Port 7 - Output data word 10
           TBEN_L4_8IOL:O.Data[108].0   // IO-Link Port 7 - Output data word 10 (INT bit0)
           TBEN_L4_8IOL:O.Data[108].1   // IO-Link Port 7 - Output data word 10 (INT bit1)
           TBEN_L4_8IOL:O.Data[108].10   // IO-Link Port 7 - Output data word 10 (INT bit10)
           TBEN_L4_8IOL:O.Data[108].11   // IO-Link Port 7 - Output data word 10 (INT bit11)
           TBEN_L4_8IOL:O.Data[108].12   // IO-Link Port 7 - Output data word 10 (INT bit12)
           TBEN_L4_8IOL:O.Data[108].13   // IO-Link Port 7 - Output data word 10 (INT bit13)
           TBEN_L4_8IOL:O.Data[108].14   // IO-Link Port 7 - Output data word 10 (INT bit14)
           TBEN_L4_8IOL:O.Data[108].15   // IO-Link Port 7 - Output data word 10 (INT bit15)
           TBEN_L4_8IOL:O.Data[108].2   // IO-Link Port 7 - Output data word 10 (INT bit2)
           TBEN_L4_8IOL:O.Data[108].3   // IO-Link Port 7 - Output data word 10 (INT bit3)
           TBEN_L4_8IOL:O.Data[108].4   // IO-Link Port 7 - Output data word 10 (INT bit4)
           TBEN_L4_8IOL:O.Data[108].5   // IO-Link Port 7 - Output data word 10 (INT bit5)
           TBEN_L4_8IOL:O.Data[108].6   // IO-Link Port 7 - Output data word 10 (INT bit6)
           TBEN_L4_8IOL:O.Data[108].7   // IO-Link Port 7 - Output data word 10 (INT bit7)
           TBEN_L4_8IOL:O.Data[108].8   // IO-Link Port 7 - Output data word 10 (INT bit8)
           TBEN_L4_8IOL:O.Data[108].9   // IO-Link Port 7 - Output data word 10 (INT bit9)
           TBEN_L4_8IOL:O.Data[109]   // IO-Link Port 7 - Output data word 11
           TBEN_L4_8IOL:O.Data[109].0   // IO-Link Port 7 - Output data word 11 (INT bit0)
           TBEN_L4_8IOL:O.Data[109].1   // IO-Link Port 7 - Output data word 11 (INT bit1)
           TBEN_L4_8IOL:O.Data[109].10   // IO-Link Port 7 - Output data word 11 (INT bit10)
           TBEN_L4_8IOL:O.Data[109].11   // IO-Link Port 7 - Output data word 11 (INT bit11)
           TBEN_L4_8IOL:O.Data[109].12   // IO-Link Port 7 - Output data word 11 (INT bit12)
           TBEN_L4_8IOL:O.Data[109].13   // IO-Link Port 7 - Output data word 11 (INT bit13)
           TBEN_L4_8IOL:O.Data[109].14   // IO-Link Port 7 - Output data word 11 (INT bit14)
           TBEN_L4_8IOL:O.Data[109].15   // IO-Link Port 7 - Output data word 11 (INT bit15)
           TBEN_L4_8IOL:O.Data[109].2   // IO-Link Port 7 - Output data word 11 (INT bit2)
           TBEN_L4_8IOL:O.Data[109].3   // IO-Link Port 7 - Output data word 11 (INT bit3)
           TBEN_L4_8IOL:O.Data[109].4   // IO-Link Port 7 - Output data word 11 (INT bit4)
           TBEN_L4_8IOL:O.Data[109].5   // IO-Link Port 7 - Output data word 11 (INT bit5)
           TBEN_L4_8IOL:O.Data[109].6   // IO-Link Port 7 - Output data word 11 (INT bit6)
           TBEN_L4_8IOL:O.Data[109].7   // IO-Link Port 7 - Output data word 11 (INT bit7)
           TBEN_L4_8IOL:O.Data[109].8   // IO-Link Port 7 - Output data word 11 (INT bit8)
           TBEN_L4_8IOL:O.Data[109].9   // IO-Link Port 7 - Output data word 11 (INT bit9)
           TBEN_L4_8IOL:O.Data[10]   // IO-Link Port 1 - Output data word 8
           TBEN_L4_8IOL:O.Data[10].0   // IO-Link Port 1 - Output data word 8 (INT bit0)
           TBEN_L4_8IOL:O.Data[10].1   // IO-Link Port 1 - Output data word 8 (INT bit1)
           TBEN_L4_8IOL:O.Data[10].10   // IO-Link Port 1 - Output data word 8 (INT bit10)
           TBEN_L4_8IOL:O.Data[10].11   // IO-Link Port 1 - Output data word 8 (INT bit11)
           TBEN_L4_8IOL:O.Data[10].12   // IO-Link Port 1 - Output data word 8 (INT bit12)
           TBEN_L4_8IOL:O.Data[10].13   // IO-Link Port 1 - Output data word 8 (INT bit13)
           TBEN_L4_8IOL:O.Data[10].14   // IO-Link Port 1 - Output data word 8 (INT bit14)
           TBEN_L4_8IOL:O.Data[10].15   // IO-Link Port 1 - Output data word 8 (INT bit15)
           TBEN_L4_8IOL:O.Data[10].2   // IO-Link Port 1 - Output data word 8 (INT bit2)
           TBEN_L4_8IOL:O.Data[10].3   // IO-Link Port 1 - Output data word 8 (INT bit3)
           TBEN_L4_8IOL:O.Data[10].4   // IO-Link Port 1 - Output data word 8 (INT bit4)
           TBEN_L4_8IOL:O.Data[10].5   // IO-Link Port 1 - Output data word 8 (INT bit5)
           TBEN_L4_8IOL:O.Data[10].6   // IO-Link Port 1 - Output data word 8 (INT bit6)
           TBEN_L4_8IOL:O.Data[10].7   // IO-Link Port 1 - Output data word 8 (INT bit7)
           TBEN_L4_8IOL:O.Data[10].8   // IO-Link Port 1 - Output data word 8 (INT bit8)
           TBEN_L4_8IOL:O.Data[10].9   // IO-Link Port 1 - Output data word 8 (INT bit9)
           TBEN_L4_8IOL:O.Data[110]   // IO-Link Port 7 - Output data word 12
           TBEN_L4_8IOL:O.Data[110].0   // IO-Link Port 7 - Output data word 12 (INT bit0)
           TBEN_L4_8IOL:O.Data[110].1   // IO-Link Port 7 - Output data word 12 (INT bit1)
           TBEN_L4_8IOL:O.Data[110].10   // IO-Link Port 7 - Output data word 12 (INT bit10)
           TBEN_L4_8IOL:O.Data[110].11   // IO-Link Port 7 - Output data word 12 (INT bit11)
           TBEN_L4_8IOL:O.Data[110].12   // IO-Link Port 7 - Output data word 12 (INT bit12)
           TBEN_L4_8IOL:O.Data[110].13   // IO-Link Port 7 - Output data word 12 (INT bit13)
           TBEN_L4_8IOL:O.Data[110].14   // IO-Link Port 7 - Output data word 12 (INT bit14)
           TBEN_L4_8IOL:O.Data[110].15   // IO-Link Port 7 - Output data word 12 (INT bit15)
           TBEN_L4_8IOL:O.Data[110].2   // IO-Link Port 7 - Output data word 12 (INT bit2)
           TBEN_L4_8IOL:O.Data[110].3   // IO-Link Port 7 - Output data word 12 (INT bit3)
           TBEN_L4_8IOL:O.Data[110].4   // IO-Link Port 7 - Output data word 12 (INT bit4)
           TBEN_L4_8IOL:O.Data[110].5   // IO-Link Port 7 - Output data word 12 (INT bit5)
           TBEN_L4_8IOL:O.Data[110].6   // IO-Link Port 7 - Output data word 12 (INT bit6)
           TBEN_L4_8IOL:O.Data[110].7   // IO-Link Port 7 - Output data word 12 (INT bit7)
           TBEN_L4_8IOL:O.Data[110].8   // IO-Link Port 7 - Output data word 12 (INT bit8)
           TBEN_L4_8IOL:O.Data[110].9   // IO-Link Port 7 - Output data word 12 (INT bit9)
           TBEN_L4_8IOL:O.Data[111]   // IO-Link Port 7 - Output data word 13
           TBEN_L4_8IOL:O.Data[111].0   // IO-Link Port 7 - Output data word 13 (INT bit0)
           TBEN_L4_8IOL:O.Data[111].1   // IO-Link Port 7 - Output data word 13 (INT bit1)
           TBEN_L4_8IOL:O.Data[111].10   // IO-Link Port 7 - Output data word 13 (INT bit10)
           TBEN_L4_8IOL:O.Data[111].11   // IO-Link Port 7 - Output data word 13 (INT bit11)
           TBEN_L4_8IOL:O.Data[111].12   // IO-Link Port 7 - Output data word 13 (INT bit12)
           TBEN_L4_8IOL:O.Data[111].13   // IO-Link Port 7 - Output data word 13 (INT bit13)
           TBEN_L4_8IOL:O.Data[111].14   // IO-Link Port 7 - Output data word 13 (INT bit14)
           TBEN_L4_8IOL:O.Data[111].15   // IO-Link Port 7 - Output data word 13 (INT bit15)
           TBEN_L4_8IOL:O.Data[111].2   // IO-Link Port 7 - Output data word 13 (INT bit2)
           TBEN_L4_8IOL:O.Data[111].3   // IO-Link Port 7 - Output data word 13 (INT bit3)
           TBEN_L4_8IOL:O.Data[111].4   // IO-Link Port 7 - Output data word 13 (INT bit4)
           TBEN_L4_8IOL:O.Data[111].5   // IO-Link Port 7 - Output data word 13 (INT bit5)
           TBEN_L4_8IOL:O.Data[111].6   // IO-Link Port 7 - Output data word 13 (INT bit6)
           TBEN_L4_8IOL:O.Data[111].7   // IO-Link Port 7 - Output data word 13 (INT bit7)
           TBEN_L4_8IOL:O.Data[111].8   // IO-Link Port 7 - Output data word 13 (INT bit8)
           TBEN_L4_8IOL:O.Data[111].9   // IO-Link Port 7 - Output data word 13 (INT bit9)
           TBEN_L4_8IOL:O.Data[112]   // IO-Link Port 7 - Output data word 14
           TBEN_L4_8IOL:O.Data[112].0   // IO-Link Port 7 - Output data word 14 (INT bit0)
           TBEN_L4_8IOL:O.Data[112].1   // IO-Link Port 7 - Output data word 14 (INT bit1)
           TBEN_L4_8IOL:O.Data[112].10   // IO-Link Port 7 - Output data word 14 (INT bit10)
           TBEN_L4_8IOL:O.Data[112].11   // IO-Link Port 7 - Output data word 14 (INT bit11)
           TBEN_L4_8IOL:O.Data[112].12   // IO-Link Port 7 - Output data word 14 (INT bit12)
           TBEN_L4_8IOL:O.Data[112].13   // IO-Link Port 7 - Output data word 14 (INT bit13)
           TBEN_L4_8IOL:O.Data[112].14   // IO-Link Port 7 - Output data word 14 (INT bit14)
           TBEN_L4_8IOL:O.Data[112].15   // IO-Link Port 7 - Output data word 14 (INT bit15)
           TBEN_L4_8IOL:O.Data[112].2   // IO-Link Port 7 - Output data word 14 (INT bit2)
           TBEN_L4_8IOL:O.Data[112].3   // IO-Link Port 7 - Output data word 14 (INT bit3)
           TBEN_L4_8IOL:O.Data[112].4   // IO-Link Port 7 - Output data word 14 (INT bit4)
           TBEN_L4_8IOL:O.Data[112].5   // IO-Link Port 7 - Output data word 14 (INT bit5)
           TBEN_L4_8IOL:O.Data[112].6   // IO-Link Port 7 - Output data word 14 (INT bit6)
           TBEN_L4_8IOL:O.Data[112].7   // IO-Link Port 7 - Output data word 14 (INT bit7)
           TBEN_L4_8IOL:O.Data[112].8   // IO-Link Port 7 - Output data word 14 (INT bit8)
           TBEN_L4_8IOL:O.Data[112].9   // IO-Link Port 7 - Output data word 14 (INT bit9)
           TBEN_L4_8IOL:O.Data[113]   // IO-Link Port 7 - Output data word 15
           TBEN_L4_8IOL:O.Data[113].0   // IO-Link Port 7 - Output data word 15 (INT bit0)
           TBEN_L4_8IOL:O.Data[113].1   // IO-Link Port 7 - Output data word 15 (INT bit1)
           TBEN_L4_8IOL:O.Data[113].10   // IO-Link Port 7 - Output data word 15 (INT bit10)
           TBEN_L4_8IOL:O.Data[113].11   // IO-Link Port 7 - Output data word 15 (INT bit11)
           TBEN_L4_8IOL:O.Data[113].12   // IO-Link Port 7 - Output data word 15 (INT bit12)
           TBEN_L4_8IOL:O.Data[113].13   // IO-Link Port 7 - Output data word 15 (INT bit13)
           TBEN_L4_8IOL:O.Data[113].14   // IO-Link Port 7 - Output data word 15 (INT bit14)
           TBEN_L4_8IOL:O.Data[113].15   // IO-Link Port 7 - Output data word 15 (INT bit15)
           TBEN_L4_8IOL:O.Data[113].2   // IO-Link Port 7 - Output data word 15 (INT bit2)
           TBEN_L4_8IOL:O.Data[113].3   // IO-Link Port 7 - Output data word 15 (INT bit3)
           TBEN_L4_8IOL:O.Data[113].4   // IO-Link Port 7 - Output data word 15 (INT bit4)
           TBEN_L4_8IOL:O.Data[113].5   // IO-Link Port 7 - Output data word 15 (INT bit5)
           TBEN_L4_8IOL:O.Data[113].6   // IO-Link Port 7 - Output data word 15 (INT bit6)
           TBEN_L4_8IOL:O.Data[113].7   // IO-Link Port 7 - Output data word 15 (INT bit7)
           TBEN_L4_8IOL:O.Data[113].8   // IO-Link Port 7 - Output data word 15 (INT bit8)
           TBEN_L4_8IOL:O.Data[113].9   // IO-Link Port 7 - Output data word 15 (INT bit9)
           TBEN_L4_8IOL:O.Data[114]   // IO-Link Port 8 - Output data word 0
           TBEN_L4_8IOL:O.Data[114].0   // IO-Link Port 8 - Output data word 0 (INT bit0)
           TBEN_L4_8IOL:O.Data[114].1   // IO-Link Port 8 - Output data word 0 (INT bit1)
           TBEN_L4_8IOL:O.Data[114].10   // IO-Link Port 8 - Output data word 0 (INT bit10)
           TBEN_L4_8IOL:O.Data[114].11   // IO-Link Port 8 - Output data word 0 (INT bit11)
           TBEN_L4_8IOL:O.Data[114].12   // IO-Link Port 8 - Output data word 0 (INT bit12)
           TBEN_L4_8IOL:O.Data[114].13   // IO-Link Port 8 - Output data word 0 (INT bit13)
           TBEN_L4_8IOL:O.Data[114].14   // IO-Link Port 8 - Output data word 0 (INT bit14)
           TBEN_L4_8IOL:O.Data[114].15   // IO-Link Port 8 - Output data word 0 (INT bit15)
           TBEN_L4_8IOL:O.Data[114].2   // IO-Link Port 8 - Output data word 0 (INT bit2)
           TBEN_L4_8IOL:O.Data[114].3   // IO-Link Port 8 - Output data word 0 (INT bit3)
           TBEN_L4_8IOL:O.Data[114].4   // IO-Link Port 8 - Output data word 0 (INT bit4)
           TBEN_L4_8IOL:O.Data[114].5   // IO-Link Port 8 - Output data word 0 (INT bit5)
           TBEN_L4_8IOL:O.Data[114].6   // IO-Link Port 8 - Output data word 0 (INT bit6)
           TBEN_L4_8IOL:O.Data[114].7   // IO-Link Port 8 - Output data word 0 (INT bit7)
           TBEN_L4_8IOL:O.Data[114].8   // IO-Link Port 8 - Output data word 0 (INT bit8)
           TBEN_L4_8IOL:O.Data[114].9   // IO-Link Port 8 - Output data word 0 (INT bit9)
           TBEN_L4_8IOL:O.Data[115]   // IO-Link Port 8 - Output data word 1
           TBEN_L4_8IOL:O.Data[115].0   // IO-Link Port 8 - Output data word 1 (INT bit0)
           TBEN_L4_8IOL:O.Data[115].1   // IO-Link Port 8 - Output data word 1 (INT bit1)
           TBEN_L4_8IOL:O.Data[115].10   // IO-Link Port 8 - Output data word 1 (INT bit10)
           TBEN_L4_8IOL:O.Data[115].11   // IO-Link Port 8 - Output data word 1 (INT bit11)
           TBEN_L4_8IOL:O.Data[115].12   // IO-Link Port 8 - Output data word 1 (INT bit12)
           TBEN_L4_8IOL:O.Data[115].13   // IO-Link Port 8 - Output data word 1 (INT bit13)
           TBEN_L4_8IOL:O.Data[115].14   // IO-Link Port 8 - Output data word 1 (INT bit14)
           TBEN_L4_8IOL:O.Data[115].15   // IO-Link Port 8 - Output data word 1 (INT bit15)
           TBEN_L4_8IOL:O.Data[115].2   // IO-Link Port 8 - Output data word 1 (INT bit2)
           TBEN_L4_8IOL:O.Data[115].3   // IO-Link Port 8 - Output data word 1 (INT bit3)
           TBEN_L4_8IOL:O.Data[115].4   // IO-Link Port 8 - Output data word 1 (INT bit4)
           TBEN_L4_8IOL:O.Data[115].5   // IO-Link Port 8 - Output data word 1 (INT bit5)
           TBEN_L4_8IOL:O.Data[115].6   // IO-Link Port 8 - Output data word 1 (INT bit6)
           TBEN_L4_8IOL:O.Data[115].7   // IO-Link Port 8 - Output data word 1 (INT bit7)
           TBEN_L4_8IOL:O.Data[115].8   // IO-Link Port 8 - Output data word 1 (INT bit8)
           TBEN_L4_8IOL:O.Data[115].9   // IO-Link Port 8 - Output data word 1 (INT bit9)
           TBEN_L4_8IOL:O.Data[116]   // IO-Link Port 8 - Output data word 2
           TBEN_L4_8IOL:O.Data[116].0   // IO-Link Port 8 - Output data word 2 (INT bit0)
           TBEN_L4_8IOL:O.Data[116].1   // IO-Link Port 8 - Output data word 2 (INT bit1)
           TBEN_L4_8IOL:O.Data[116].10   // IO-Link Port 8 - Output data word 2 (INT bit10)
           TBEN_L4_8IOL:O.Data[116].11   // IO-Link Port 8 - Output data word 2 (INT bit11)
           TBEN_L4_8IOL:O.Data[116].12   // IO-Link Port 8 - Output data word 2 (INT bit12)
           TBEN_L4_8IOL:O.Data[116].13   // IO-Link Port 8 - Output data word 2 (INT bit13)
           TBEN_L4_8IOL:O.Data[116].14   // IO-Link Port 8 - Output data word 2 (INT bit14)
           TBEN_L4_8IOL:O.Data[116].15   // IO-Link Port 8 - Output data word 2 (INT bit15)
           TBEN_L4_8IOL:O.Data[116].2   // IO-Link Port 8 - Output data word 2 (INT bit2)
           TBEN_L4_8IOL:O.Data[116].3   // IO-Link Port 8 - Output data word 2 (INT bit3)
           TBEN_L4_8IOL:O.Data[116].4   // IO-Link Port 8 - Output data word 2 (INT bit4)
           TBEN_L4_8IOL:O.Data[116].5   // IO-Link Port 8 - Output data word 2 (INT bit5)
           TBEN_L4_8IOL:O.Data[116].6   // IO-Link Port 8 - Output data word 2 (INT bit6)
           TBEN_L4_8IOL:O.Data[116].7   // IO-Link Port 8 - Output data word 2 (INT bit7)
           TBEN_L4_8IOL:O.Data[116].8   // IO-Link Port 8 - Output data word 2 (INT bit8)
           TBEN_L4_8IOL:O.Data[116].9   // IO-Link Port 8 - Output data word 2 (INT bit9)
           TBEN_L4_8IOL:O.Data[117]   // IO-Link Port 8 - Output data word 3
           TBEN_L4_8IOL:O.Data[117].0   // IO-Link Port 8 - Output data word 3 (INT bit0)
           TBEN_L4_8IOL:O.Data[117].1   // IO-Link Port 8 - Output data word 3 (INT bit1)
           TBEN_L4_8IOL:O.Data[117].10   // IO-Link Port 8 - Output data word 3 (INT bit10)
           TBEN_L4_8IOL:O.Data[117].11   // IO-Link Port 8 - Output data word 3 (INT bit11)
           TBEN_L4_8IOL:O.Data[117].12   // IO-Link Port 8 - Output data word 3 (INT bit12)
           TBEN_L4_8IOL:O.Data[117].13   // IO-Link Port 8 - Output data word 3 (INT bit13)
           TBEN_L4_8IOL:O.Data[117].14   // IO-Link Port 8 - Output data word 3 (INT bit14)
           TBEN_L4_8IOL:O.Data[117].15   // IO-Link Port 8 - Output data word 3 (INT bit15)
           TBEN_L4_8IOL:O.Data[117].2   // IO-Link Port 8 - Output data word 3 (INT bit2)
           TBEN_L4_8IOL:O.Data[117].3   // IO-Link Port 8 - Output data word 3 (INT bit3)
           TBEN_L4_8IOL:O.Data[117].4   // IO-Link Port 8 - Output data word 3 (INT bit4)
           TBEN_L4_8IOL:O.Data[117].5   // IO-Link Port 8 - Output data word 3 (INT bit5)
           TBEN_L4_8IOL:O.Data[117].6   // IO-Link Port 8 - Output data word 3 (INT bit6)
           TBEN_L4_8IOL:O.Data[117].7   // IO-Link Port 8 - Output data word 3 (INT bit7)
           TBEN_L4_8IOL:O.Data[117].8   // IO-Link Port 8 - Output data word 3 (INT bit8)
           TBEN_L4_8IOL:O.Data[117].9   // IO-Link Port 8 - Output data word 3 (INT bit9)
           TBEN_L4_8IOL:O.Data[118]   // IO-Link Port 8 - Output data word 4
           TBEN_L4_8IOL:O.Data[118].0   // IO-Link Port 8 - Output data word 4 (INT bit0)
           TBEN_L4_8IOL:O.Data[118].1   // IO-Link Port 8 - Output data word 4 (INT bit1)
           TBEN_L4_8IOL:O.Data[118].10   // IO-Link Port 8 - Output data word 4 (INT bit10)
           TBEN_L4_8IOL:O.Data[118].11   // IO-Link Port 8 - Output data word 4 (INT bit11)
           TBEN_L4_8IOL:O.Data[118].12   // IO-Link Port 8 - Output data word 4 (INT bit12)
           TBEN_L4_8IOL:O.Data[118].13   // IO-Link Port 8 - Output data word 4 (INT bit13)
           TBEN_L4_8IOL:O.Data[118].14   // IO-Link Port 8 - Output data word 4 (INT bit14)
           TBEN_L4_8IOL:O.Data[118].15   // IO-Link Port 8 - Output data word 4 (INT bit15)
           TBEN_L4_8IOL:O.Data[118].2   // IO-Link Port 8 - Output data word 4 (INT bit2)
           TBEN_L4_8IOL:O.Data[118].3   // IO-Link Port 8 - Output data word 4 (INT bit3)
           TBEN_L4_8IOL:O.Data[118].4   // IO-Link Port 8 - Output data word 4 (INT bit4)
           TBEN_L4_8IOL:O.Data[118].5   // IO-Link Port 8 - Output data word 4 (INT bit5)
           TBEN_L4_8IOL:O.Data[118].6   // IO-Link Port 8 - Output data word 4 (INT bit6)
           TBEN_L4_8IOL:O.Data[118].7   // IO-Link Port 8 - Output data word 4 (INT bit7)
           TBEN_L4_8IOL:O.Data[118].8   // IO-Link Port 8 - Output data word 4 (INT bit8)
           TBEN_L4_8IOL:O.Data[118].9   // IO-Link Port 8 - Output data word 4 (INT bit9)
           TBEN_L4_8IOL:O.Data[119]   // IO-Link Port 8 - Output data word 5
           TBEN_L4_8IOL:O.Data[119].0   // IO-Link Port 8 - Output data word 5 (INT bit0)
           TBEN_L4_8IOL:O.Data[119].1   // IO-Link Port 8 - Output data word 5 (INT bit1)
           TBEN_L4_8IOL:O.Data[119].10   // IO-Link Port 8 - Output data word 5 (INT bit10)
           TBEN_L4_8IOL:O.Data[119].11   // IO-Link Port 8 - Output data word 5 (INT bit11)
           TBEN_L4_8IOL:O.Data[119].12   // IO-Link Port 8 - Output data word 5 (INT bit12)
           TBEN_L4_8IOL:O.Data[119].13   // IO-Link Port 8 - Output data word 5 (INT bit13)
           TBEN_L4_8IOL:O.Data[119].14   // IO-Link Port 8 - Output data word 5 (INT bit14)
           TBEN_L4_8IOL:O.Data[119].15   // IO-Link Port 8 - Output data word 5 (INT bit15)
           TBEN_L4_8IOL:O.Data[119].2   // IO-Link Port 8 - Output data word 5 (INT bit2)
           TBEN_L4_8IOL:O.Data[119].3   // IO-Link Port 8 - Output data word 5 (INT bit3)
           TBEN_L4_8IOL:O.Data[119].4   // IO-Link Port 8 - Output data word 5 (INT bit4)
           TBEN_L4_8IOL:O.Data[119].5   // IO-Link Port 8 - Output data word 5 (INT bit5)
           TBEN_L4_8IOL:O.Data[119].6   // IO-Link Port 8 - Output data word 5 (INT bit6)
           TBEN_L4_8IOL:O.Data[119].7   // IO-Link Port 8 - Output data word 5 (INT bit7)
           TBEN_L4_8IOL:O.Data[119].8   // IO-Link Port 8 - Output data word 5 (INT bit8)
           TBEN_L4_8IOL:O.Data[119].9   // IO-Link Port 8 - Output data word 5 (INT bit9)
           TBEN_L4_8IOL:O.Data[11]   // IO-Link Port 1 - Output data word 9
           TBEN_L4_8IOL:O.Data[11].0   // IO-Link Port 1 - Output data word 9 (INT bit0)
           TBEN_L4_8IOL:O.Data[11].1   // IO-Link Port 1 - Output data word 9 (INT bit1)
           TBEN_L4_8IOL:O.Data[11].10   // IO-Link Port 1 - Output data word 9 (INT bit10)
           TBEN_L4_8IOL:O.Data[11].11   // IO-Link Port 1 - Output data word 9 (INT bit11)
           TBEN_L4_8IOL:O.Data[11].12   // IO-Link Port 1 - Output data word 9 (INT bit12)
           TBEN_L4_8IOL:O.Data[11].13   // IO-Link Port 1 - Output data word 9 (INT bit13)
           TBEN_L4_8IOL:O.Data[11].14   // IO-Link Port 1 - Output data word 9 (INT bit14)
           TBEN_L4_8IOL:O.Data[11].15   // IO-Link Port 1 - Output data word 9 (INT bit15)
           TBEN_L4_8IOL:O.Data[11].2   // IO-Link Port 1 - Output data word 9 (INT bit2)
           TBEN_L4_8IOL:O.Data[11].3   // IO-Link Port 1 - Output data word 9 (INT bit3)
           TBEN_L4_8IOL:O.Data[11].4   // IO-Link Port 1 - Output data word 9 (INT bit4)
           TBEN_L4_8IOL:O.Data[11].5   // IO-Link Port 1 - Output data word 9 (INT bit5)
           TBEN_L4_8IOL:O.Data[11].6   // IO-Link Port 1 - Output data word 9 (INT bit6)
           TBEN_L4_8IOL:O.Data[11].7   // IO-Link Port 1 - Output data word 9 (INT bit7)
           TBEN_L4_8IOL:O.Data[11].8   // IO-Link Port 1 - Output data word 9 (INT bit8)
           TBEN_L4_8IOL:O.Data[11].9   // IO-Link Port 1 - Output data word 9 (INT bit9)
           TBEN_L4_8IOL:O.Data[120]   // IO-Link Port 8 - Output data word 6
           TBEN_L4_8IOL:O.Data[120].0   // IO-Link Port 8 - Output data word 6 (INT bit0)
           TBEN_L4_8IOL:O.Data[120].1   // IO-Link Port 8 - Output data word 6 (INT bit1)
           TBEN_L4_8IOL:O.Data[120].10   // IO-Link Port 8 - Output data word 6 (INT bit10)
           TBEN_L4_8IOL:O.Data[120].11   // IO-Link Port 8 - Output data word 6 (INT bit11)
           TBEN_L4_8IOL:O.Data[120].12   // IO-Link Port 8 - Output data word 6 (INT bit12)
           TBEN_L4_8IOL:O.Data[120].13   // IO-Link Port 8 - Output data word 6 (INT bit13)
           TBEN_L4_8IOL:O.Data[120].14   // IO-Link Port 8 - Output data word 6 (INT bit14)
           TBEN_L4_8IOL:O.Data[120].15   // IO-Link Port 8 - Output data word 6 (INT bit15)
           TBEN_L4_8IOL:O.Data[120].2   // IO-Link Port 8 - Output data word 6 (INT bit2)
           TBEN_L4_8IOL:O.Data[120].3   // IO-Link Port 8 - Output data word 6 (INT bit3)
           TBEN_L4_8IOL:O.Data[120].4   // IO-Link Port 8 - Output data word 6 (INT bit4)
           TBEN_L4_8IOL:O.Data[120].5   // IO-Link Port 8 - Output data word 6 (INT bit5)
           TBEN_L4_8IOL:O.Data[120].6   // IO-Link Port 8 - Output data word 6 (INT bit6)
           TBEN_L4_8IOL:O.Data[120].7   // IO-Link Port 8 - Output data word 6 (INT bit7)
           TBEN_L4_8IOL:O.Data[120].8   // IO-Link Port 8 - Output data word 6 (INT bit8)
           TBEN_L4_8IOL:O.Data[120].9   // IO-Link Port 8 - Output data word 6 (INT bit9)
           TBEN_L4_8IOL:O.Data[121]   // IO-Link Port 8 - Output data word 7
           TBEN_L4_8IOL:O.Data[121].0   // IO-Link Port 8 - Output data word 7 (INT bit0)
           TBEN_L4_8IOL:O.Data[121].1   // IO-Link Port 8 - Output data word 7 (INT bit1)
           TBEN_L4_8IOL:O.Data[121].10   // IO-Link Port 8 - Output data word 7 (INT bit10)
           TBEN_L4_8IOL:O.Data[121].11   // IO-Link Port 8 - Output data word 7 (INT bit11)
           TBEN_L4_8IOL:O.Data[121].12   // IO-Link Port 8 - Output data word 7 (INT bit12)
           TBEN_L4_8IOL:O.Data[121].13   // IO-Link Port 8 - Output data word 7 (INT bit13)
           TBEN_L4_8IOL:O.Data[121].14   // IO-Link Port 8 - Output data word 7 (INT bit14)
           TBEN_L4_8IOL:O.Data[121].15   // IO-Link Port 8 - Output data word 7 (INT bit15)
           TBEN_L4_8IOL:O.Data[121].2   // IO-Link Port 8 - Output data word 7 (INT bit2)
           TBEN_L4_8IOL:O.Data[121].3   // IO-Link Port 8 - Output data word 7 (INT bit3)
           TBEN_L4_8IOL:O.Data[121].4   // IO-Link Port 8 - Output data word 7 (INT bit4)
